LIN {X 0,Y 520.436,Z 843.44,A -85,B 0,C 180,E1 4700.36,E2 4700.36} C_VEL
LIN {X 0,Y 520.239,Z 843.44,A -85,B 0,C 180,E1 4705.948,E2 4705.948} C_VEL
LIN {X 0,Y 520.311,Z 843.44,A -85,B 0,C 180,E1 4711.467,E2 4711.467} C_VEL
LIN {X 0,Y 520.266,Z 843.44,A -85,B 0,C 180,E1 4717.522,E2 4717.522} C_VEL
LIN {X 0,Y 520.062,Z 843.44,A -85,B 0,C 180,E1 4723.497,E2 4723.497} C_VEL
LIN {X 0,Y 520.261,Z 843.44,A -85,B 0,C 180,E1 4730.087,E2 4730.087} C_VEL
LIN {X 0,Y 524.81,Z 853.402,A -85,B 0,C 180,E1 4730.693,E2 4730.693} C_VEL
LIN {X 0,Y 537.138,Z 878.782,A -85,B 0,C 180,E1 4732.342,E2 4732.342} C_VEL
LIN {X 0,Y 535.242,Z 919.42,A -85,B 0,C 180,E1 4733.697,E2 4733.697} C_VEL
LIN {X 0,Y 532.879,Z 957.32,A -85,B 0,C 180,E1 4735.589,E2 4735.589} C_VEL
LIN {X 0,Y 530.11,Z 994.748,A -85,B 0,C 180,E1 4738.147,E2 4738.147} C_VEL
LIN {X 0,Y 527.279,Z 1030.228,A -85,B 0,C 180,E1 4741.356,E2 4741.356} C_VEL
LIN {X 0,Y 524.799,Z 1061.7,A -85,B 0,C 180,E1 4745.046,E2 4745.046} C_VEL
LIN {X 0,Y 522.926,Z 1089.588,A -85,B 0,C 180,E1 4749.298,E2 4749.298} C_VEL
LIN {X 0,Y 521.748,Z 1111.144,A -85,B 0,C 180,E1 4753.621,E2 4753.621} C_VEL
LIN {X 0,Y 521.215,Z 1128.039,A -85,B 0,C 180,E1 4758.307,E2 4758.307} C_VEL
LIN {X 0,Y 520.97,Z 1138.048,A -85,B 0,C 180,E1 4762.51,E2 4762.51} C_VEL
LIN {X 0,Y 520.916,Z 1143.672,A -85,B 0,C 180,E1 4766.678,E2 4766.678} C_VEL
LIN {X 0,Y 521.004,Z 1144.637,A -85,B 0,C 180,E1 4771.66,E2 4771.66} C_VEL
LIN {X 0,Y 520.954,Z 1140.667,A -85,B 0,C 180,E1 4775.819,E2 4775.819} C_VEL
LIN {X 0,Y 521.037,Z 1132.292,A -85,B 0,C 180,E1 4780.049,E2 4780.049} C_VEL
LIN {X 0,Y 521.477,Z 1118.445,A -85,B 0,C 180,E1 4784.459,E2 4784.459} C_VEL
LIN {X 0,Y 522.247,Z 1099.604,A -85,B 0,C 180,E1 4788.751,E2 4788.751} C_VEL
LIN {X 0,Y 523.772,Z 1076.177,A -85,B 0,C 180,E1 4792.795,E2 4792.795} C_VEL
LIN {X 0,Y 525.898,Z 1047.674,A -85,B 0,C 180,E1 4796.619,E2 4796.619} C_VEL
LIN {X 0,Y 528.516,Z 1014.37,A -85,B 0,C 180,E1 4800.095,E2 4800.095} C_VEL
LIN {X 0,Y 531.435,Z 977.699,A -85,B 0,C 180,E1 4803.023,E2 4803.023} C_VEL
LIN {X 0,Y 534.228,Z 938.21,A -85,B 0,C 180,E1 4805.358,E2 4805.358} C_VEL
LIN {X 0,Y 536.423,Z 897.49,A -85,B 0,C 180,E1 4807.024,E2 4807.024} C_VEL
LIN {X 0,Y 536.641,Z 877.029,A -85,B 0,C 180,E1 4807.655,E2 4807.655} C_VEL
LIN {X 0,Y 520.249,Z 844.875,A -85,B 0,C 180,E1 4809.787,E2 4809.787} C_VEL
LIN {X 0,Y 520.083,Z 843.44,A -85,B 0,C 180,E1 4809.907,E2 4809.907} C_VEL
LIN {X 0,Y 520.164,Z 843.44,A -85,B 0,C 180,E1 4815.876,E2 4815.876} C_VEL
LIN {X 0,Y 520.179,Z 843.44,A -85,B 0,C 180,E1 4821.559,E2 4821.559} C_VEL
LIN {X 0,Y 520.166,Z 843.44,A -85,B 0,C 180,E1 4827.277,E2 4827.277} C_VEL
LIN {X 0,Y 520.251,Z 843.44,A -85,B 0,C 180,E1 4832.35,E2 4832.35} C_VEL
LIN {X 0,Y 520.43,Z 843.44,A -85,B 0,C 180,E1 4838.103,E2 4838.103} C_VEL
LIN {X 0,Y 520.561,Z 843.44,A -85,B 0,C 180,E1 4843.15,E2 4843.15} C_VEL
LIN {X 0,Y 520.576,Z 843.44,A -85,B 0,C 180,E1 4848.293,E2 4848.293} C_VEL
LIN {X 0,Y 520.63,Z 843.44,A -85,B 0,C 180,E1 4853.343,E2 4853.343} C_VEL
LIN {X 0,Y 520.641,Z 843.44,A -85,B 0,C 180,E1 4858.339,E2 4858.339} C_VEL
LIN {X 0,Y 520.67,Z 843.44,A -85,B 0,C 180,E1 4863.323,E2 4863.323} C_VEL
LIN {X 0,Y 520.537,Z 843.44,A -85,B 0,C 180,E1 4868.334,E2 4868.334} C_VEL
LIN {X 0,Y 520.491,Z 843.44,A -85,B 0,C 180,E1 4873.411,E2 4873.411} C_VEL
LIN {X 0,Y 520.432,Z 843.44,A -85,B 0,C 180,E1 4878.599,E2 4878.599} C_VEL
LIN {X 0,Y 520.333,Z 843.44,A -85,B 0,C 180,E1 4883.954,E2 4883.954} C_VEL
LIN {X 0,Y 520.209,Z 843.44,A -85,B 0,C 180,E1 4889.546,E2 4889.546} C_VEL
LIN {X 0,Y 520.065,Z 843.44,A -85,B 0,C 180,E1 4894.185,E2 4894.185} C_VEL
LIN {X 0,Y 516.099,Z 843.44,A -85,B 0,C 180,E1 4896.07,E2 4896.07} C_VEL
LIN {X 0,Y 512.255,Z 843.44,A -85,B 0,C 180,E1 4897.985,E2 4897.985} C_VEL
LIN {X 0,Y 512.25,Z 843.44,A -85,B 0,C 180,E1 4902.65,E2 4902.65} C_VEL
LIN {X 0,Y 512.2,Z 843.929,A -85,B 0,C 180,E1 4908.861,E2 4908.861} C_VEL
LIN {X 0,Y 531.6,Z 881.961,A -85,B 0,C 180,E1 4911.305,E2 4911.305} C_VEL
LIN {X 0,Y 530.037,Z 926.984,A -85,B 0,C 180,E1 4912.388,E2 4912.388} C_VEL
LIN {X 0,Y 527.526,Z 969.74,A -85,B 0,C 180,E1 4914.165,E2 4914.165} C_VEL
LIN {X 0,Y 524.424,Z 1009.394,A -85,B 0,C 180,E1 4916.557,E2 4916.557} C_VEL
LIN {X 0,Y 521.221,Z 1047.334,A -85,B 0,C 180,E1 4919.68,E2 4919.68} C_VEL
LIN {X 0,Y 518.367,Z 1080.674,A -85,B 0,C 180,E1 4923.286,E2 4923.286} C_VEL
LIN {X 0,Y 515.864,Z 1110.299,A -85,B 0,C 180,E1 4927.446,E2 4927.446} C_VEL
LIN {X 0,Y 514.329,Z 1134.904,A -85,B 0,C 180,E1 4932.009,E2 4932.009} C_VEL
LIN {X 0,Y 513.485,Z 1152.465,A -85,B 0,C 180,E1 4936.403,E2 4936.403} C_VEL
LIN {X 0,Y 513.102,Z 1164.64,A -85,B 0,C 180,E1 4940.764,E2 4940.764} C_VEL
LIN {X 0,Y 512.92,Z 1171.926,A -85,B 0,C 180,E1 4944.937,E2 4944.937} C_VEL
LIN {X 0,Y 512.92,Z 1174.659,A -85,B 0,C 180,E1 4948.314,E2 4948.314} C_VEL
LIN {X 0,Y 513.175,Z 1174.659,A -85,B 0,C 180,E1 4951.685,E2 4951.685} C_VEL
LIN {X 0,Y 513.034,Z 1169.517,A -85,B 0,C 180,E1 4956.757,E2 4956.757} C_VEL
LIN {X 0,Y 513.348,Z 1159.09,A -85,B 0,C 180,E1 4961.445,E2 4961.445} C_VEL
LIN {X 0,Y 513.978,Z 1142.713,A -85,B 0,C 180,E1 4966.196,E2 4966.196} C_VEL
LIN {X 0,Y 515.2,Z 1121.769,A -85,B 0,C 180,E1 4970.578,E2 4970.578} C_VEL
LIN {X 0,Y 517.007,Z 1095.883,A -85,B 0,C 180,E1 4974.708,E2 4974.708} C_VEL
LIN {X 0,Y 519.533,Z 1066.104,A -85,B 0,C 180,E1 4978.4,E2 4978.4} C_VEL
LIN {X 0,Y 522.495,Z 1031.765,A -85,B 0,C 180,E1 4981.709,E2 4981.709} C_VEL
LIN {X 0,Y 525.589,Z 994.442,A -85,B 0,C 180,E1 4984.44,E2 4984.44} C_VEL
LIN {X 0,Y 528.55,Z 952.967,A -85,B 0,C 180,E1 4986.629,E2 4986.629} C_VEL
LIN {X 0,Y 530.862,Z 909.195,A -85,B 0,C 180,E1 4988.126,E2 4988.126} C_VEL
LIN {X 0,Y 531.26,Z 880.332,A -85,B 0,C 180,E1 4988.755,E2 4988.755} C_VEL
LIN {X 0,Y 512.197,Z 843.964,A -85,B 0,C 180,E1 4991.138,E2 4991.138} C_VEL
LIN {X 0,Y 512.246,Z 843.44,A -85,B 0,C 180,E1 4997.432,E2 4997.432} C_VEL
LIN {X 0,Y 512.233,Z 843.44,A -85,B 0,C 180,E1 5002.694,E2 5002.694} C_VEL
LIN {X 0,Y 512.289,Z 843.44,A -85,B 0,C 180,E1 5008.675,E2 5008.675} C_VEL
LIN {X 0,Y 512.351,Z 843.44,A -85,B 0,C 180,E1 5013.783,E2 5013.783} C_VEL
LIN {X 0,Y 512.551,Z 843.44,A -85,B 0,C 180,E1 5019.312,E2 5019.312} C_VEL
LIN {X 0,Y 512.462,Z 843.44,A -85,B 0,C 180,E1 5024.633,E2 5024.633} C_VEL
LIN {X 0,Y 512.632,Z 843.44,A -85,B 0,C 180,E1 5029.827,E2 5029.827} C_VEL
LIN {X 0,Y 512.845,Z 843.44,A -85,B 0,C 180,E1 5034.936,E2 5034.936} C_VEL
LIN {X 0,Y 512.86,Z 843.44,A -85,B 0,C 180,E1 5040,E2 5040} C_VEL
LIN {X 0,Y 512.812,Z 843.44,A -85,B 0,C 180,E1 5045.064,E2 5045.064} C_VEL
LIN {X 0,Y 512.698,Z 843.44,A -85,B 0,C 180,E1 5050.171,E2 5050.171} C_VEL
LIN {X 0,Y 512.592,Z 843.44,A -85,B 0,C 180,E1 5055.363,E2 5055.363} C_VEL
LIN {X 0,Y 512.532,Z 843.44,A -85,B 0,C 180,E1 5060.689,E2 5060.689} C_VEL
LIN {X 0,Y 512.323,Z 843.44,A -85,B 0,C 180,E1 5066.218,E2 5066.218} C_VEL
LIN {X 0,Y 512.445,Z 843.44,A -85,B 0,C 180,E1 5072.007,E2 5072.007} C_VEL
LIN {X 0,Y 512.324,Z 843.44,A -85,B 0,C 180,E1 5078.208,E2 5078.208} C_VEL
LIN {X 0,Y 512.131,Z 843.44,A -85,B 0,C 180,E1 5085.002,E2 5085.002} C_VEL
LIN {X 0,Y 512.276,Z 843.444,A -85,B 0,C 180,E1 5089.342,E2 5089.342} C_VEL
LIN {X 0,Y 514.638,Z 849.042,A -85,B 0,C 180,E1 5089.67,E2 5089.67} C_VEL
LIN {X 0,Y 530.839,Z 880.706,A -85,B 0,C 180,E1 5091.868,E2 5091.868} C_VEL
LIN {X 0,Y 528.596,Z 923.315,A -85,B 0,C 180,E1 5093.345,E2 5093.345} C_VEL
LIN {X 0,Y 525.764,Z 963.463,A -85,B 0,C 180,E1 5095.463,E2 5095.463} C_VEL
LIN {X 0,Y 522.824,Z 998.946,A -85,B 0,C 180,E1 5098.021,E2 5098.021} C_VEL
LIN {X 0,Y 519.772,Z 1033.362,A -85,B 0,C 180,E1 5101.259,E2 5101.259} C_VEL
LIN {X 0,Y 517.213,Z 1063.294,A -85,B 0,C 180,E1 5104.884,E2 5104.884} C_VEL
LIN {X 0,Y 515.23,Z 1089.586,A -85,B 0,C 180,E1 5108.975,E2 5108.975} C_VEL
LIN {X 0,Y 513.952,Z 1111.142,A -85,B 0,C 180,E1 5113.365,E2 5113.365} C_VEL
LIN {X 0,Y 513.334,Z 1128.036,A -85,B 0,C 180,E1 5118.125,E2 5118.125} C_VEL
LIN {X 0,Y 513.063,Z 1138.047,A -85,B 0,C 180,E1 5122.394,E2 5122.394} C_VEL
LIN {X 0,Y 513.014,Z 1143.671,A -85,B 0,C 180,E1 5126.627,E2 5126.627} C_VEL
LIN {X 0,Y 513.108,Z 1144.638,A -85,B 0,C 180,E1 5131.685,E2 5131.685} C_VEL
LIN {X 0,Y 513.059,Z 1140.668,A -85,B 0,C 180,E1 5135.908,E2 5135.908} C_VEL
LIN {X 0,Y 513.159,Z 1132.409,A -85,B 0,C 180,E1 5140.162,E2 5140.162} C_VEL
LIN {X 0,Y 513.614,Z 1118.479,A -85,B 0,C 180,E1 5144.677,E2 5144.677} C_VEL
LIN {X 0,Y 514.451,Z 1100.693,A -85,B 0,C 180,E1 5148.824,E2 5148.824} C_VEL
LIN {X 0,Y 516.145,Z 1077.203,A -85,B 0,C 180,E1 5152.991,E2 5152.991} C_VEL
LIN {X 0,Y 518.466,Z 1048.615,A -85,B 0,C 180,E1 5156.917,E2 5156.917} C_VEL
LIN {X 0,Y 521.362,Z 1015.638,A -85,B 0,C 180,E1 5160.431,E2 5160.431} C_VEL
LIN {X 0,Y 524.602,Z 978.202,A -85,B 0,C 180,E1 5163.473,E2 5163.473} C_VEL
LIN {X 0,Y 527.627,Z 938.991,A -85,B 0,C 180,E1 5165.826,E2 5165.826} C_VEL
LIN {X 0,Y 530.015,Z 898.735,A -85,B 0,C 180,E1 5167.5,E2 5167.5} C_VEL
LIN {X 0,Y 530.326,Z 880.119,A -85,B 0,C 180,E1 5168.102,E2 5168.102} C_VEL
LIN {X 0,Y 512.171,Z 843.949,A -85,B 0,C 180,E1 5170.568,E2 5170.568} C_VEL
LIN {X 0,Y 512.214,Z 843.44,A -85,B 0,C 180,E1 5175.007,E2 5175.007} C_VEL
LIN {X 0,Y 512.272,Z 843.44,A -85,B 0,C 180,E1 5179.986,E2 5179.986} C_VEL
LIN {X 0,Y 512.175,Z 843.44,A -85,B 0,C 180,E1 5185.96,E2 5185.96} C_VEL
LIN {X 0,Y 512.31,Z 843.44,A -85,B 0,C 180,E1 5192.086,E2 5192.086} C_VEL
LIN {X 0,Y 512.445,Z 843.44,A -85,B 0,C 180,E1 5197.493,E2 5197.493} C_VEL
LIN {X 0,Y 512.652,Z 843.44,A -85,B 0,C 180,E1 5202.882,E2 5202.882} C_VEL
LIN {X 0,Y 512.665,Z 843.44,A -85,B 0,C 180,E1 5208.11,E2 5208.11} C_VEL
LIN {X 0,Y 512.72,Z 843.44,A -85,B 0,C 180,E1 5213.24,E2 5213.24} C_VEL
LIN {X 0,Y 512.741,Z 843.44,A -85,B 0,C 180,E1 5218.314,E2 5218.314} C_VEL
LIN {X 0,Y 512.775,Z 843.44,A -85,B 0,C 180,E1 5223.374,E2 5223.374} C_VEL
LIN {X 0,Y 512.632,Z 843.44,A -85,B 0,C 180,E1 5228.464,E2 5228.464} C_VEL
LIN {X 0,Y 512.577,Z 843.44,A -85,B 0,C 180,E1 5233.709,E2 5233.709} C_VEL
LIN {X 0,Y 512.486,Z 843.44,A -85,B 0,C 180,E1 5239.569,E2 5239.569} C_VEL
LIN {X 0,Y 512.383,Z 843.44,A -85,B 0,C 180,E1 5244.349,E2 5244.349} C_VEL
LIN {X 0,Y 512.246,Z 843.44,A -85,B 0,C 180,E1 5250.052,E2 5250.052} C_VEL
LIN {X 0,Y 512.205,Z 843.44,A -85,B 0,C 180,E1 5256.1,E2 5256.1} C_VEL
LIN {X 0,Y 512.255,Z 843.44,A -85,B 0,C 180,E1 5257.985,E2 5257.985} C_VEL
LIN {X 0,Y 509.802,Z 843.44,A -85,B 0,C 180,E1 5259.415,E2 5259.415} C_VEL
LIN {X 0,Y 504.24,Z 843.44,A -85,B 0,C 180,E1 5261.805,E2 5261.805} C_VEL
LIN {X 0,Y 504.315,Z 844.166,A -85,B 0,C 180,E1 5268.086,E2 5268.086} C_VEL
LIN {X 0,Y 525.368,Z 884.453,A -85,B 0,C 180,E1 5270.809,E2 5270.809} C_VEL
LIN {X 0,Y 523.699,Z 927.636,A -85,B 0,C 180,E1 5271.878,E2 5271.878} C_VEL
LIN {X 0,Y 521.018,Z 969.675,A -85,B 0,C 180,E1 5273.643,E2 5273.643} C_VEL
LIN {X 0,Y 517.667,Z 1009.395,A -85,B 0,C 180,E1 5276.062,E2 5276.062} C_VEL
LIN {X 0,Y 514.143,Z 1047.323,A -85,B 0,C 180,E1 5279.217,E2 5279.217} C_VEL
LIN {X 0,Y 510.953,Z 1081.461,A -85,B 0,C 180,E1 5282.973,E2 5282.973} C_VEL
LIN {X 0,Y 508.335,Z 1110.222,A -85,B 0,C 180,E1 5287.079,E2 5287.079} C_VEL
LIN {X 0,Y 506.689,Z 1134.088,A -85,B 0,C 180,E1 5291.542,E2 5291.542} C_VEL
LIN {X 0,Y 505.667,Z 1152.464,A -85,B 0,C 180,E1 5296.188,E2 5296.188} C_VEL
LIN {X 0,Y 505.21,Z 1165.116,A -85,B 0,C 180,E1 5300.834,E2 5300.834} C_VEL
LIN {X 0,Y 505.022,Z 1171.926,A -85,B 0,C 180,E1 5304.857,E2 5304.857} C_VEL
LIN {X 0,Y 505.018,Z 1174.659,A -85,B 0,C 180,E1 5308.288,E2 5308.288} C_VEL
LIN {X 0,Y 505.27,Z 1174.659,A -85,B 0,C 180,E1 5311.712,E2 5311.712} C_VEL
LIN {X 0,Y 505.137,Z 1169.517,A -85,B 0,C 180,E1 5316.863,E2 5316.863} C_VEL
LIN {X 0,Y 505.471,Z 1159.091,A -85,B 0,C 180,E1 5321.626,E2 5321.626} C_VEL
LIN {X 0,Y 506.178,Z 1142.714,A -85,B 0,C 180,E1 5326.452,E2 5326.452} C_VEL
LIN {X 0,Y 507.529,Z 1121.768,A -85,B 0,C 180,E1 5330.903,E2 5330.903} C_VEL
LIN {X 0,Y 509.494,Z 1096.45,A -85,B 0,C 180,E1 5335.014,E2 5335.014} C_VEL
LIN {X 0,Y 512.269,Z 1066.678,A -85,B 0,C 180,E1 5338.774,E2 5338.774} C_VEL
LIN {X 0,Y 515.521,Z 1032.556,A -85,B 0,C 180,E1 5342.118,E2 5342.118} C_VEL
LIN {X 0,Y 518.902,Z 994.749,A -85,B 0,C 180,E1 5344.927,E2 5344.927} C_VEL
LIN {X 0,Y 522.128,Z 953.443,A -85,B 0,C 180,E1 5347.133,E2 5347.133} C_VEL
LIN {X 0,Y 524.58,Z 911.065,A -85,B 0,C 180,E1 5348.614,E2 5348.614} C_VEL
LIN {X 0,Y 525.023,Z 883.051,A -85,B 0,C 180,E1 5349.25,E2 5349.25} C_VEL
LIN {X 0,Y 504.318,Z 844.136,A -85,B 0,C 180,E1 5351.914,E2 5351.914} C_VEL
LIN {X 0,Y 504.266,Z 843.44,A -85,B 0,C 180,E1 5358.428,E2 5358.428} C_VEL
LIN {X 0,Y 504.343,Z 843.44,A -85,B 0,C 180,E1 5363.887,E2 5363.887} C_VEL
LIN {X 0,Y 504.327,Z 843.44,A -85,B 0,C 180,E1 5370.195,E2 5370.195} C_VEL
LIN {X 0,Y 504.428,Z 843.44,A -85,B 0,C 180,E1 5375.241,E2 5375.241} C_VEL
LIN {X 0,Y 504.669,Z 843.44,A -85,B 0,C 180,E1 5380.798,E2 5380.798} C_VEL
LIN {X 0,Y 504.482,Z 843.44,A -85,B 0,C 180,E1 5386.155,E2 5386.155} C_VEL
LIN {X 0,Y 504.712,Z 843.44,A -85,B 0,C 180,E1 5391.403,E2 5391.403} C_VEL
LIN {X 0,Y 504.875,Z 843.44,A -85,B 0,C 180,E1 5396.573,E2 5396.573} C_VEL
LIN {X 0,Y 504.845,Z 843.44,A -85,B 0,C 180,E1 5401.713,E2 5401.713} C_VEL
LIN {X 0,Y 504.804,Z 843.44,A -85,B 0,C 180,E1 5406.867,E2 5406.867} C_VEL
LIN {X 0,Y 504.723,Z 843.44,A -85,B 0,C 180,E1 5412.08,E2 5412.08} C_VEL
LIN {X 0,Y 504.677,Z 843.44,A -85,B 0,C 180,E1 5417.397,E2 5417.397} C_VEL
LIN {X 0,Y 504.507,Z 843.44,A -85,B 0,C 180,E1 5422.881,E2 5422.881} C_VEL
LIN {X 0,Y 504.393,Z 843.44,A -85,B 0,C 180,E1 5428.598,E2 5428.598} C_VEL
LIN {X 0,Y 504.487,Z 843.44,A -85,B 0,C 180,E1 5434.632,E2 5434.632} C_VEL
LIN {X 0,Y 504.225,Z 843.44,A -85,B 0,C 180,E1 5441.176,E2 5441.176} C_VEL
LIN {X 0,Y 504.16,Z 843.44,A -85,B 0,C 180,E1 5446.495,E2 5446.495} C_VEL
LIN {X 0,Y 504.287,Z 843.585,A -85,B 0,C 180,E1 5448.555,E2 5448.555} C_VEL
LIN {X 0,Y 508.488,Z 852.603,A -85,B 0,C 180,E1 5449.143,E2 5449.143} C_VEL
LIN {X 0,Y 524.313,Z 883.255,A -85,B 0,C 180,E1 5451.391,E2 5451.391} C_VEL
LIN {X 0,Y 522.069,Z 925.289,A -85,B 0,C 180,E1 5452.909,E2 5452.909} C_VEL
LIN {X 0,Y 518.814,Z 967.192,A -85,B 0,C 180,E1 5455.193,E2 5455.193} C_VEL
LIN {X 0,Y 515.224,Z 1006.042,A -85,B 0,C 180,E1 5458.139,E2 5458.139} C_VEL
LIN {X 0,Y 511.93,Z 1040.776,A -85,B 0,C 180,E1 5461.641,E2 5461.641} C_VEL
LIN {X 0,Y 509.114,Z 1071.581,A -85,B 0,C 180,E1 5465.688,E2 5465.688} C_VEL
LIN {X 0,Y 507.049,Z 1097.701,A -85,B 0,C 180,E1 5470.181,E2 5470.181} C_VEL
LIN {X 0,Y 505.926,Z 1117.481,A -85,B 0,C 180,E1 5474.719,E2 5474.719} C_VEL
LIN {X 0,Y 505.31,Z 1132.641,A -85,B 0,C 180,E1 5479.678,E2 5479.678} C_VEL
LIN {X 0,Y 505.091,Z 1140.795,A -85,B 0,C 180,E1 5483.998,E2 5483.998} C_VEL
LIN {X 0,Y 505.025,Z 1144.675,A -85,B 0,C 180,E1 5488.288,E2 5488.288} C_VEL
LIN {X 0,Y 505.202,Z 1144.638,A -85,B 0,C 180,E1 5491.711,E2 5491.711} C_VEL
LIN {X 0,Y 505.165,Z 1140.668,A -85,B 0,C 180,E1 5496.001,E2 5496.001} C_VEL
LIN {X 0,Y 505.276,Z 1132.411,A -85,B 0,C 180,E1 5500.322,E2 5500.322} C_VEL
LIN {X 0,Y 505.793,Z 1118.22,A -85,B 0,C 180,E1 5504.984,E2 5504.984} C_VEL
LIN {X 0,Y 506.723,Z 1100.695,A -85,B 0,C 180,E1 5509.122,E2 5509.122} C_VEL
LIN {X 0,Y 508.535,Z 1077.437,A -85,B 0,C 180,E1 5513.319,E2 5513.319} C_VEL
LIN {X 0,Y 511.181,Z 1047.883,A -85,B 0,C 180,E1 5517.425,E2 5517.425} C_VEL
LIN {X 0,Y 514.461,Z 1014.39,A -85,B 0,C 180,E1 5521.007,E2 5521.007} C_VEL
LIN {X 0,Y 517.927,Z 977.123,A -85,B 0,C 180,E1 5524.045,E2 5524.045} C_VEL
LIN {X 0,Y 521.224,Z 937.756,A -85,B 0,C 180,E1 5526.405,E2 5526.405} C_VEL
LIN {X 0,Y 523.809,Z 897.766,A -85,B 0,C 180,E1 5528.062,E2 5528.062} C_VEL
LIN {X 0,Y 523.988,Z 883.073,A -85,B 0,C 180,E1 5528.553,E2 5528.553} C_VEL
LIN {X 0,Y 504.309,Z 844.705,A -85,B 0,C 180,E1 5531.332,E2 5531.332} C_VEL
LIN {X 0,Y 504.227,Z 843.44,A -85,B 0,C 180,E1 5531.404,E2 5531.404} C_VEL
LIN {X 0,Y 504.232,Z 843.44,A -85,B 0,C 180,E1 5536.505,E2 5536.505} C_VEL
LIN {X 0,Y 504.326,Z 843.44,A -85,B 0,C 180,E1 5541.074,E2 5541.074} C_VEL
LIN {X 0,Y 504.262,Z 843.44,A -85,B 0,C 180,E1 5547.41,E2 5547.41} C_VEL
LIN {X 0,Y 504.434,Z 843.44,A -85,B 0,C 180,E1 5553.825,E2 5553.825} C_VEL
LIN {X 0,Y 504.603,Z 843.44,A -85,B 0,C 180,E1 5558.971,E2 5558.971} C_VEL
LIN {X 0,Y 504.748,Z 843.44,A -85,B 0,C 180,E1 5564.392,E2 5564.392} C_VEL
LIN {X 0,Y 504.775,Z 843.44,A -85,B 0,C 180,E1 5570.584,E2 5570.584} C_VEL
LIN {X 0,Y 505.018,Z 843.44,A -85,B 0,C 180,E1 5576.574,E2 5576.574} C_VEL
LIN {X 0,Y 505.117,Z 843.44,A -85,B 0,C 180,E1 5581.712,E2 5581.712} C_VEL
LIN {X 0,Y 504.887,Z 843.44,A -85,B 0,C 180,E1 5586.866,E2 5586.866} C_VEL
LIN {X 0,Y 504.71,Z 843.44,A -85,B 0,C 180,E1 5592.08,E2 5592.08} C_VEL
LIN {X 0,Y 504.634,Z 843.44,A -85,B 0,C 180,E1 5597.399,E2 5597.399} C_VEL
LIN {X 0,Y 504.495,Z 843.44,A -85,B 0,C 180,E1 5602.882,E2 5602.882} C_VEL
LIN {X 0,Y 504.363,Z 843.44,A -85,B 0,C 180,E1 5608.6,E2 5608.6} C_VEL
LIN {X 0,Y 504.27,Z 843.44,A -85,B 0,C 180,E1 5614.649,E2 5614.649} C_VEL
LIN {X 0,Y 504.286,Z 843.44,A -85,B 0,C 180,E1 5621.17,E2 5621.17} C_VEL
LIN {X 0,Y 504.24,Z 843.44,A -85,B 0,C 180,E1 5621.805,E2 5621.805} C_VEL
LIN {X 0,Y 500.248,Z 843.44,A -85,B 0,C 180,E1 5623.754,E2 5623.754} C_VEL
LIN {X 0,Y 496.309,Z 843.44,A -85,B 0,C 180,E1 5625.732,E2 5625.732} C_VEL
LIN {X 0,Y 496.36,Z 843.44,A -85,B 0,C 180,E1 5627.23,E2 5627.23} C_VEL
LIN {X 0,Y 500.68,Z 852.873,A -85,B 0,C 180,E1 5627.879,E2 5627.879} C_VEL
LIN {X 0,Y 519.189,Z 886.645,A -85,B 0,C 180,E1 5630.297,E2 5630.297} C_VEL
LIN {X 0,Y 517.346,Z 929.486,A -85,B 0,C 180,E1 5631.4,E2 5631.4} C_VEL
LIN {X 0,Y 514.459,Z 970.757,A -85,B 0,C 180,E1 5633.17,E2 5633.17} C_VEL
LIN {X 0,Y 510.866,Z 1010.222,A -85,B 0,C 180,E1 5635.615,E2 5635.615} C_VEL
LIN {X 0,Y 507.025,Z 1048.058,A -85,B 0,C 180,E1 5638.816,E2 5638.816} C_VEL
LIN {X 0,Y 503.561,Z 1082.165,A -85,B 0,C 180,E1 5642.64,E2 5642.64} C_VEL
LIN {X 0,Y 500.669,Z 1111.503,A -85,B 0,C 180,E1 5646.932,E2 5646.932} C_VEL
LIN {X 0,Y 498.866,Z 1135.122,A -85,B 0,C 180,E1 5651.482,E2 5651.482} C_VEL
LIN {X 0,Y 497.845,Z 1152.463,A -85,B 0,C 180,E1 5655.967,E2 5655.967} C_VEL
LIN {X 0,Y 497.339,Z 1165.116,A -85,B 0,C 180,E1 5660.687,E2 5660.687} C_VEL
LIN {X 0,Y 497.129,Z 1171.926,A -85,B 0,C 180,E1 5664.775,E2 5664.775} C_VEL
LIN {X 0,Y 497.116,Z 1174.659,A -85,B 0,C 180,E1 5668.261,E2 5668.261} C_VEL
LIN {X 0,Y 497.38,Z 1174.659,A -85,B 0,C 180,E1 5671.739,E2 5671.739} C_VEL
LIN {X 0,Y 497.246,Z 1169.517,A -85,B 0,C 180,E1 5676.973,E2 5676.973} C_VEL
LIN {X 0,Y 497.593,Z 1159.092,A -85,B 0,C 180,E1 5681.812,E2 5681.812} C_VEL
LIN {X 0,Y 498.373,Z 1142.716,A -85,B 0,C 180,E1 5686.717,E2 5686.717} C_VEL
LIN {X 0,Y 499.845,Z 1121.766,A -85,B 0,C 180,E1 5691.24,E2 5691.24} C_VEL
LIN {X 0,Y 502.127,Z 1095.85,A -85,B 0,C 180,E1 5695.497,E2 5695.497} C_VEL
LIN {X 0,Y 505.19,Z 1065.52,A -85,B 0,C 180,E1 5699.352,E2 5699.352} C_VEL
LIN {X 0,Y 508.683,Z 1032.016,A -85,B 0,C 180,E1 5702.652,E2 5702.652} C_VEL
LIN {X 0,Y 512.396,Z 993.619,A -85,B 0,C 180,E1 5705.515,E2 5705.515} C_VEL
LIN {X 0,Y 515.79,Z 953.429,A -85,B 0,C 180,E1 5707.669,E2 5707.669} C_VEL
LIN {X 0,Y 518.472,Z 909.512,A -85,B 0,C 180,E1 5709.2,E2 5709.2} C_VEL
LIN {X 0,Y 518.709,Z 885.753,A -85,B 0,C 180,E1 5709.765,E2 5709.765} C_VEL
LIN {X 0,Y 496.486,Z 844.831,A -85,B 0,C 180,E1 5712.71,E2 5712.71} C_VEL
LIN {X 0,Y 496.36,Z 843.44,A -85,B 0,C 180,E1 5712.845,E2 5712.845} C_VEL
LIN {X 0,Y 496.321,Z 843.44,A -85,B 0,C 180,E1 5718.021,E2 5718.021} C_VEL
LIN {X 0,Y 496.379,Z 843.44,A -85,B 0,C 180,E1 5724.719,E2 5724.719} C_VEL
LIN {X 0,Y 496.428,Z 843.44,A -85,B 0,C 180,E1 5730.9,E2 5730.9} C_VEL
LIN {X 0,Y 496.541,Z 843.44,A -85,B 0,C 180,E1 5736.73,E2 5736.73} C_VEL
LIN {X 0,Y 496.767,Z 843.44,A -85,B 0,C 180,E1 5742.317,E2 5742.317} C_VEL
LIN {X 0,Y 496.779,Z 843.44,A -85,B 0,C 180,E1 5749.499,E2 5749.499} C_VEL
LIN {X 0,Y 497.034,Z 843.44,A -85,B 0,C 180,E1 5754.774,E2 5754.774} C_VEL
LIN {X 0,Y 497.066,Z 843.44,A -85,B 0,C 180,E1 5760,E2 5760} C_VEL
LIN {X 0,Y 496.998,Z 843.44,A -85,B 0,C 180,E1 5765.226,E2 5765.226} C_VEL
LIN {X 0,Y 496.862,Z 843.44,A -85,B 0,C 180,E1 5770.499,E2 5770.499} C_VEL
LIN {X 0,Y 496.752,Z 843.44,A -85,B 0,C 180,E1 5775.866,E2 5775.866} C_VEL
LIN {X 0,Y 496.65,Z 843.44,A -85,B 0,C 180,E1 5781.382,E2 5781.382} C_VEL
LIN {X 0,Y 496.453,Z 843.44,A -85,B 0,C 180,E1 5787.124,E2 5787.124} C_VEL
LIN {X 0,Y 496.556,Z 843.44,A -85,B 0,C 180,E1 5793.161,E2 5793.161} C_VEL
LIN {X 0,Y 496.352,Z 843.44,A -85,B 0,C 180,E1 5799.674,E2 5799.674} C_VEL
LIN {X 0,Y 496.237,Z 843.44,A -85,B 0,C 180,E1 5805.62,E2 5805.62} C_VEL
LIN {X 0,Y 496.296,Z 843.44,A -85,B 0,C 180,E1 5807.709,E2 5807.709} C_VEL
LIN {X 0,Y 498.826,Z 849.175,A -85,B 0,C 180,E1 5808.101,E2 5808.101} C_VEL
LIN {X 0,Y 517.933,Z 886.118,A -85,B 0,C 180,E1 5810.924,E2 5810.924} C_VEL
LIN {X 0,Y 515.588,Z 926.528,A -85,B 0,C 180,E1 5812.431,E2 5812.431} C_VEL
LIN {X 0,Y 512.245,Z 966.564,A -85,B 0,C 180,E1 5814.634,E2 5814.634} C_VEL
LIN {X 0,Y 508.414,Z 1005.256,A -85,B 0,C 180,E1 5817.583,E2 5817.583} C_VEL
LIN {X 0,Y 504.691,Z 1040.94,A -85,B 0,C 180,E1 5821.219,E2 5821.219} C_VEL
LIN {X 0,Y 501.599,Z 1071.754,A -85,B 0,C 180,E1 5825.328,E2 5825.328} C_VEL
LIN {X 0,Y 499.447,Z 1096.508,A -85,B 0,C 180,E1 5829.616,E2 5829.616} C_VEL
LIN {X 0,Y 498.163,Z 1116.36,A -85,B 0,C 180,E1 5834.179,E2 5834.179} C_VEL
LIN {X 0,Y 497.497,Z 1131.501,A -85,B 0,C 180,E1 5839.072,E2 5839.072} C_VEL
LIN {X 0,Y 497.231,Z 1139.586,A -85,B 0,C 180,E1 5843.027,E2 5843.027} C_VEL
LIN {X 0,Y 497.207,Z 1143.67,A -85,B 0,C 180,E1 5846.52,E2 5846.52} C_VEL
LIN {X 0,Y 497.296,Z 1144.639,A -85,B 0,C 180,E1 5851.739,E2 5851.739} C_VEL
LIN {X 0,Y 497.257,Z 1140.669,A -85,B 0,C 180,E1 5856.097,E2 5856.097} C_VEL
LIN {X 0,Y 497.382,Z 1132.412,A -85,B 0,C 180,E1 5860.488,E2 5860.488} C_VEL
LIN {X 0,Y 498.002,Z 1117.708,A -85,B 0,C 180,E1 5865.374,E2 5865.374} C_VEL
LIN {X 0,Y 499.265,Z 1098.01,A -85,B 0,C 180,E1 5869.987,E2 5869.987} C_VEL
LIN {X 0,Y 501.513,Z 1072.667,A -85,B 0,C 180,E1 5874.439,E2 5874.439} C_VEL
LIN {X 0,Y 504.374,Z 1043.677,A -85,B 0,C 180,E1 5878.362,E2 5878.362} C_VEL
LIN {X 0,Y 507.811,Z 1010.756,A -85,B 0,C 180,E1 5881.821,E2 5881.821} C_VEL
LIN {X 0,Y 511.322,Z 976.201,A -85,B 0,C 180,E1 5884.617,E2 5884.617} C_VEL
LIN {X 0,Y 514.775,Z 937.841,A -85,B 0,C 180,E1 5886.932,E2 5886.932} C_VEL
LIN {X 0,Y 517.534,Z 898.37,A -85,B 0,C 180,E1 5888.584,E2 5888.584} C_VEL
LIN {X 0,Y 517.651,Z 886.086,A -85,B 0,C 180,E1 5889.012,E2 5889.012} C_VEL
LIN {X 0,Y 498.819,Z 849.224,A -85,B 0,C 180,E1 5891.809,E2 5891.809} C_VEL
LIN {X 0,Y 496.227,Z 843.44,A -85,B 0,C 180,E1 5892.287,E2 5892.287} C_VEL
LIN {X 0,Y 496.302,Z 843.44,A -85,B 0,C 180,E1 5898.019,E2 5898.019} C_VEL
LIN {X 0,Y 496.367,Z 843.44,A -85,B 0,C 180,E1 5904.718,E2 5904.718} C_VEL
LIN {X 0,Y 496.417,Z 843.44,A -85,B 0,C 180,E1 5910.899,E2 5910.899} C_VEL
LIN {X 0,Y 496.539,Z 843.44,A -85,B 0,C 180,E1 5916.73,E2 5916.73} C_VEL
LIN {X 0,Y 496.776,Z 843.44,A -85,B 0,C 180,E1 5922.317,E2 5922.317} C_VEL
LIN {X 0,Y 496.844,Z 843.44,A -85,B 0,C 180,E1 5927.726,E2 5927.726} C_VEL
LIN {X 0,Y 496.924,Z 843.44,A -85,B 0,C 180,E1 5933.024,E2 5933.024} C_VEL
LIN {X 0,Y 496.964,Z 843.44,A -85,B 0,C 180,E1 5938.26,E2 5938.26} C_VEL
LIN {X 0,Y 496.986,Z 843.44,A -85,B 0,C 180,E1 5943.482,E2 5943.482} C_VEL
LIN {X 0,Y 496.824,Z 843.44,A -85,B 0,C 180,E1 5948.735,E2 5948.735} C_VEL
LIN {X 0,Y 496.767,Z 843.44,A -85,B 0,C 180,E1 5954.064,E2 5954.064} C_VEL
LIN {X 0,Y 496.64,Z 843.44,A -85,B 0,C 180,E1 5959.624,E2 5959.624} C_VEL
LIN {X 0,Y 496.528,Z 843.44,A -85,B 0,C 180,E1 5965.18,E2 5965.18} C_VEL
LIN {X 0,Y 496.321,Z 843.44,A -85,B 0,C 180,E1 5971.646,E2 5971.646} C_VEL
LIN {X 0,Y 496.32,Z 843.44,A -85,B 0,C 180,E1 5977.768,E2 5977.768} C_VEL
LIN {X 0,Y 496.339,Z 843.44,A -85,B 0,C 180,E1 5984.366,E2 5984.366} C_VEL
LIN {X 0,Y 496.309,Z 843.44,A -85,B 0,C 180,E1 5985.732,E2 5985.732} C_VEL
LIN {X 0,Y 496.515,Z 846.56,A -85,B 0,C 180,E1 5986.618,E2 5986.618} C_VEL
LIN {X 0,Y 498.004,Z 857.238,A -85,B 0,C 180,E1 5987.561,E2 5987.561} C_VEL
LIN {X 0,Y 502.24,Z 869.127,A -85,B 0,C 180,E1 5988.343,E2 5988.343} C_VEL
LIN {X 0,Y 512.968,Z 889.52,A -85,B 0,C 180,E1 5989.786,E2 5989.786} C_VEL
LIN {X 0,Y 511.021,Z 931.258,A -85,B 0,C 180,E1 5990.91,E2 5990.91} C_VEL
LIN {X 0,Y 507.989,Z 971.227,A -85,B 0,C 180,E1 5992.651,E2 5992.651} C_VEL
LIN {X 0,Y 504.009,Z 1011.681,A -85,B 0,C 180,E1 5995.204,E2 5995.204} C_VEL
LIN {X 0,Y 500.106,Z 1047.572,A -85,B 0,C 180,E1 5998.282,E2 5998.282} C_VEL
LIN {X 0,Y 496.283,Z 1081.676,A -85,B 0,C 180,E1 6002.136,E2 6002.136} C_VEL
LIN {X 0,Y 493.282,Z 1110.168,A -85,B 0,C 180,E1 6006.327,E2 6006.327} C_VEL
LIN {X 0,Y 491.224,Z 1134.139,A -85,B 0,C 180,E1 6010.95,E2 6010.95} C_VEL
LIN {X 0,Y 490.037,Z 1152.462,A -85,B 0,C 180,E1 6015.738,E2 6015.738} C_VEL
LIN {X 0,Y 489.447,Z 1165.24,A -85,B 0,C 180,E1 6020.594,E2 6020.594} C_VEL
LIN {X 0,Y 489.233,Z 1171.926,A -85,B 0,C 180,E1 6024.691,E2 6024.691} C_VEL
LIN {X 0,Y 489.214,Z 1174.659,A -85,B 0,C 180,E1 6028.233,E2 6028.233} C_VEL
LIN {X 0,Y 489.474,Z 1174.659,A -85,B 0,C 180,E1 6031.767,E2 6031.767} C_VEL
LIN {X 0,Y 489.349,Z 1169.517,A -85,B 0,C 180,E1 6037.086,E2 6037.086} C_VEL
LIN {X 0,Y 489.72,Z 1159.092,A -85,B 0,C 180,E1 6042.005,E2 6042.005} C_VEL
LIN {X 0,Y 490.561,Z 1143.355,A -85,B 0,C 180,E1 6046.824,E2 6046.824} C_VEL
LIN {X 0,Y 492.107,Z 1122.841,A -85,B 0,C 180,E1 6051.379,E2 6051.379} C_VEL
LIN {X 0,Y 494.561,Z 1097.332,A -85,B 0,C 180,E1 6055.69,E2 6055.69} C_VEL
LIN {X 0,Y 497.806,Z 1067.903,A -85,B 0,C 180,E1 6059.546,E2 6059.546} C_VEL
LIN {X 0,Y 501.774,Z 1032.527,A -85,B 0,C 180,E1 6063.112,E2 6063.112} C_VEL
LIN {X 0,Y 505.741,Z 994.713,A -85,B 0,C 180,E1 6065.978,E2 6065.978} C_VEL
LIN {X 0,Y 509.493,Z 953.43,A -85,B 0,C 180,E1 6068.218,E2 6068.218} C_VEL
LIN {X 0,Y 512.333,Z 909.284,A -85,B 0,C 180,E1 6069.762,E2 6069.762} C_VEL
LIN {X 0,Y 512.56,Z 888.801,A -85,B 0,C 180,E1 6070.268,E2 6070.268} C_VEL
LIN {X 0,Y 490.006,Z 848.156,A -85,B 0,C 180,E1 6073.342,E2 6073.342} C_VEL
LIN {X 0,Y 488.401,Z 843.44,A -85,B 0,C 180,E1 6073.66,E2 6073.66} C_VEL
LIN {X 0,Y 488.421,Z 843.44,A -85,B 0,C 180,E1 6079.55,E2 6079.55} C_VEL
LIN {X 0,Y 488.439,Z 843.44,A -85,B 0,C 180,E1 6086.215,E2 6086.215} C_VEL
LIN {X 0,Y 488.519,Z 843.44,A -85,B 0,C 180,E1 6092.398,E2 6092.398} C_VEL
LIN {X 0,Y 488.697,Z 843.44,A -85,B 0,C 180,E1 6098.252,E2 6098.252} C_VEL
LIN {X 0,Y 488.758,Z 843.44,A -85,B 0,C 180,E1 6103.867,E2 6103.867} C_VEL
LIN {X 0,Y 488.856,Z 843.44,A -85,B 0,C 180,E1 6109.327,E2 6109.327} C_VEL
LIN {X 0,Y 489.121,Z 843.44,A -85,B 0,C 180,E1 6114.689,E2 6114.689} C_VEL
LIN {X 0,Y 489.165,Z 843.44,A -85,B 0,C 180,E1 6120,E2 6120} C_VEL
LIN {X 0,Y 489.083,Z 843.44,A -85,B 0,C 180,E1 6125.311,E2 6125.311} C_VEL
LIN {X 0,Y 488.936,Z 843.44,A -85,B 0,C 180,E1 6130.671,E2 6130.671} C_VEL
LIN {X 0,Y 488.784,Z 843.44,A -85,B 0,C 180,E1 6136.851,E2 6136.851} C_VEL
LIN {X 0,Y 488.673,Z 843.44,A -85,B 0,C 180,E1 6142.12,E2 6142.12} C_VEL
LIN {X 0,Y 488.536,Z 843.44,A -85,B 0,C 180,E1 6147.601,E2 6147.601} C_VEL
LIN {X 0,Y 488.614,Z 843.44,A -85,B 0,C 180,E1 6153.771,E2 6153.771} C_VEL
LIN {X 0,Y 488.435,Z 843.44,A -85,B 0,C 180,E1 6159.432,E2 6159.432} C_VEL
LIN {X 0,Y 488.331,Z 843.44,A -85,B 0,C 180,E1 6165.292,E2 6165.292} C_VEL
LIN {X 0,Y 488.371,Z 843.44,A -85,B 0,C 180,E1 6166.84,E2 6166.84} C_VEL
LIN {X 0,Y 490.891,Z 849.214,A -85,B 0,C 180,E1 6167.258,E2 6167.258} C_VEL
LIN {X 0,Y 510.151,Z 885.647,A -85,B 0,C 180,E1 6170.185,E2 6170.185} C_VEL
LIN {X 0,Y 511.746,Z 890.75,A -85,B 0,C 180,E1 6170.515,E2 6170.515} C_VEL
LIN {X 0,Y 508.956,Z 929.535,A -85,B 0,C 180,E1 6172.023,E2 6172.023} C_VEL
LIN {X 0,Y 505.396,Z 969.044,A -85,B 0,C 180,E1 6174.275,E2 6174.275} C_VEL
LIN {X 0,Y 501.385,Z 1006.478,A -85,B 0,C 180,E1 6177.197,E2 6177.197} C_VEL
LIN {X 0,Y 497.437,Z 1041.136,A -85,B 0,C 180,E1 6180.785,E2 6180.785} C_VEL
LIN {X 0,Y 494.124,Z 1071.751,A -85,B 0,C 180,E1 6184.929,E2 6184.929} C_VEL
LIN {X 0,Y 491.681,Z 1097.666,A -85,B 0,C 180,E1 6189.527,E2 6189.527} C_VEL
LIN {X 0,Y 490.274,Z 1118.012,A -85,B 0,C 180,E1 6194.376,E2 6194.376} C_VEL
LIN {X 0,Y 489.577,Z 1132.637,A -85,B 0,C 180,E1 6199.342,E2 6199.342} C_VEL
LIN {X 0,Y 489.3,Z 1140.792,A -85,B 0,C 180,E1 6203.803,E2 6203.803} C_VEL
LIN {X 0,Y 489.221,Z 1144.675,A -85,B 0,C 180,E1 6208.232,E2 6208.232} C_VEL
LIN {X 0,Y 489.39,Z 1144.639,A -85,B 0,C 180,E1 6211.767,E2 6211.767} C_VEL
LIN {X 0,Y 489.347,Z 1140.67,A -85,B 0,C 180,E1 6216.196,E2 6216.196} C_VEL
LIN {X 0,Y 489.516,Z 1132.414,A -85,B 0,C 180,E1 6220.659,E2 6220.659} C_VEL
LIN {X 0,Y 490.102,Z 1119.254,A -85,B 0,C 180,E1 6225.172,E2 6225.172} C_VEL
LIN {X 0,Y 491.229,Z 1101.781,A -85,B 0,C 180,E1 6229.516,E2 6229.516} C_VEL
LIN {X 0,Y 493.401,Z 1078.489,A -85,B 0,C 180,E1 6233.906,E2 6233.906} C_VEL
LIN {X 0,Y 496.62,Z 1048.52,A -85,B 0,C 180,E1 6238.219,E2 6238.219} C_VEL
LIN {X 0,Y 500.374,Z 1015.549,A -85,B 0,C 180,E1 6241.865,E2 6241.865} C_VEL
LIN {X 0,Y 504.476,Z 978.114,A -85,B 0,C 180,E1 6245.008,E2 6245.008} C_VEL
LIN {X 0,Y 508.401,Z 937.767,A -85,B 0,C 180,E1 6247.479,E2 6247.479} C_VEL
LIN {X 0,Y 511.347,Z 898.929,A -85,B 0,C 180,E1 6249.123,E2 6249.123} C_VEL
LIN {X 0,Y 511.28,Z 888.929,A -85,B 0,C 180,E1 6249.503,E2 6249.503} C_VEL
LIN {X 0,Y 493.856,Z 854.553,A -85,B 0,C 180,E1 6252.221,E2 6252.221} C_VEL
LIN {X 0,Y 488.387,Z 844.171,A -85,B 0,C 180,E1 6253.026,E2 6253.026} C_VEL
LIN {X 0,Y 488.397,Z 843.44,A -85,B 0,C 180,E1 6257.862,E2 6257.862} C_VEL
LIN {X 0,Y 488.378,Z 843.44,A -85,B 0,C 180,E1 6264.052,E2 6264.052} C_VEL
LIN {X 0,Y 488.442,Z 843.44,A -85,B 0,C 180,E1 6270.377,E2 6270.377} C_VEL
LIN {X 0,Y 488.636,Z 843.44,A -85,B 0,C 180,E1 6276.331,E2 6276.331} C_VEL
LIN {X 0,Y 488.845,Z 843.44,A -85,B 0,C 180,E1 6282.021,E2 6282.021} C_VEL
LIN {X 0,Y 488.97,Z 843.44,A -85,B 0,C 180,E1 6287.525,E2 6287.525} C_VEL
LIN {X 0,Y 489.01,Z 843.44,A -85,B 0,C 180,E1 6292.91,E2 6292.91} C_VEL
LIN {X 0,Y 489.064,Z 843.44,A -85,B 0,C 180,E1 6298.232,E2 6298.232} C_VEL
LIN {X 0,Y 489.08,Z 843.44,A -85,B 0,C 180,E1 6303.538,E2 6303.538} C_VEL
LIN {X 0,Y 488.914,Z 843.44,A -85,B 0,C 180,E1 6309.008,E2 6309.008} C_VEL
LIN {X 0,Y 488.829,Z 843.44,A -85,B 0,C 180,E1 6314.297,E2 6314.297} C_VEL
LIN {X 0,Y 488.731,Z 843.44,A -85,B 0,C 180,E1 6319.854,E2 6319.854} C_VEL
LIN {X 0,Y 488.565,Z 843.44,A -85,B 0,C 180,E1 6325.62,E2 6325.62} C_VEL
LIN {X 0,Y 488.418,Z 843.44,A -85,B 0,C 180,E1 6331.683,E2 6331.683} C_VEL
LIN {X 0,Y 488.403,Z 843.44,A -85,B 0,C 180,E1 6338.164,E2 6338.164} C_VEL
LIN {X 0,Y 488.417,Z 843.44,A -85,B 0,C 180,E1 6344.716,E2 6344.716} C_VEL
LIN {X 0,Y 488.426,Z 843.44,A -85,B 0,C 180,E1 6346.378,E2 6346.378} C_VEL
LIN {X 0,Y 490.81,Z 849.095,A -85,B 0,C 180,E1 6346.765,E2 6346.765} C_VEL
LIN {X 0,Y 502.24,Z 869.127,A -85,B 0,C 180,E1 6348.343,E2 6348.343} C_VEL
LIN {X 0,Y 506.135,Z 880.489,A -85,B 0,C 180,E1 6348.939,E2 6348.939} C_VEL
LIN {X 0,Y 506.48,Z 902.56,A -85,B 0,C 180,E1 6349.502,E2 6349.502} C_VEL
LIN {X 0,Y 504.044,Z 942.331,A -85,B 0,C 180,E1 6350.762,E2 6350.762} C_VEL
LIN {X 0,Y 500.696,Z 981.834,A -85,B 0,C 180,E1 6352.694,E2 6352.694} C_VEL
LIN {X 0,Y 496.377,Z 1020.467,A -85,B 0,C 180,E1 6355.354,E2 6355.354} C_VEL
LIN {X 0,Y 491.967,Z 1057.531,A -85,B 0,C 180,E1 6358.816,E2 6358.816} C_VEL
LIN {X 0,Y 488.046,Z 1090.045,A -85,B 0,C 180,E1 6362.822,E2 6362.822} C_VEL
LIN {X 0,Y 484.836,Z 1118.607,A -85,B 0,C 180,E1 6367.439,E2 6367.439} C_VEL
LIN {X 0,Y 482.893,Z 1141.028,A -85,B 0,C 180,E1 6372.278,E2 6372.278} C_VEL
LIN {X 0,Y 481.875,Z 1157.894,A -85,B 0,C 180,E1 6377.338,E2 6377.338} C_VEL
LIN {X 0,Y 481.493,Z 1167.965,A -85,B 0,C 180,E1 6381.893,E2 6381.893} C_VEL
LIN {X 0,Y 481.381,Z 1173.637,A -85,B 0,C 180,E1 6386.406,E2 6386.406} C_VEL
LIN {X 0,Y 481.589,Z 1174.659,A -85,B 0,C 180,E1 6391.796,E2 6391.796} C_VEL
LIN {X 0,Y 481.47,Z 1169.517,A -85,B 0,C 180,E1 6397.202,E2 6397.202} C_VEL
LIN {X 0,Y 481.863,Z 1159.093,A -85,B 0,C 180,E1 6402.204,E2 6402.204} C_VEL
LIN {X 0,Y 482.758,Z 1143.624,A -85,B 0,C 180,E1 6407.031,E2 6407.031} C_VEL
LIN {X 0,Y 484.428,Z 1123.467,A -85,B 0,C 180,E1 6411.609,E2 6411.609} C_VEL
LIN {X 0,Y 487.13,Z 1097.644,A -85,B 0,C 180,E1 6416.062,E2 6416.062} C_VEL
LIN {X 0,Y 490.74,Z 1067.209,A -85,B 0,C 180,E1 6420.099,E2 6420.099} C_VEL
LIN {X 0,Y 494.961,Z 1032.68,A -85,B 0,C 180,E1 6423.613,E2 6423.613} C_VEL
LIN {X 0,Y 499.305,Z 993.913,A -85,B 0,C 180,E1 6426.573,E2 6426.573} C_VEL
LIN {X 0,Y 503.244,Z 952.671,A -85,B 0,C 180,E1 6428.803,E2 6428.803} C_VEL
LIN {X 0,Y 506.177,Z 910.447,A -85,B 0,C 180,E1 6430.301,E2 6430.301} C_VEL
LIN {X 0,Y 506.494,Z 891.83,A -85,B 0,C 180,E1 6430.779,E2 6430.779} C_VEL
LIN {X 0,Y 482.863,Z 849.068,A -85,B 0,C 180,E1 6434.121,E2 6434.121} C_VEL
LIN {X 0,Y 480.518,Z 843.44,A -85,B 0,C 180,E1 6434.593,E2 6434.593} C_VEL
LIN {X 0,Y 480.5,Z 843.44,A -85,B 0,C 180,E1 6441.091,E2 6441.091} C_VEL
LIN {X 0,Y 480.506,Z 843.44,A -85,B 0,C 180,E1 6447.733,E2 6447.733} C_VEL
LIN {X 0,Y 480.645,Z 843.44,A -85,B 0,C 180,E1 6453.927,E2 6453.927} C_VEL
LIN {X 0,Y 480.883,Z 843.44,A -85,B 0,C 180,E1 6460.289,E2 6460.289} C_VEL
LIN {X 0,Y 480.75,Z 843.44,A -85,B 0,C 180,E1 6466.669,E2 6466.669} C_VEL
LIN {X 0,Y 481.151,Z 843.44,A -85,B 0,C 180,E1 6472.793,E2 6472.793} C_VEL
LIN {X 0,Y 481.429,Z 843.44,A -85,B 0,C 180,E1 6478.204,E2 6478.204} C_VEL
LIN {X 0,Y 481.304,Z 843.44,A -85,B 0,C 180,E1 6483.595,E2 6483.595} C_VEL
LIN {X 0,Y 481.1,Z 843.44,A -85,B 0,C 180,E1 6489.022,E2 6489.022} C_VEL
LIN {X 0,Y 480.975,Z 843.44,A -85,B 0,C 180,E1 6494.535,E2 6494.535} C_VEL
LIN {X 0,Y 480.824,Z 843.44,A -85,B 0,C 180,E1 6500.194,E2 6500.194} C_VEL
LIN {X 0,Y 480.641,Z 843.44,A -85,B 0,C 180,E1 6506.073,E2 6506.073} C_VEL
LIN {X 0,Y 480.662,Z 843.44,A -85,B 0,C 180,E1 6512.255,E2 6512.255} C_VEL
LIN {X 0,Y 480.609,Z 843.44,A -85,B 0,C 180,E1 6518.284,E2 6518.284} C_VEL
LIN {X 0,Y 480.431,Z 843.44,A -85,B 0,C 180,E1 6524.667,E2 6524.667} C_VEL
LIN {X 0,Y 480.436,Z 843.44,A -85,B 0,C 180,E1 6525.947,E2 6525.947} C_VEL
LIN {X 0,Y 482.833,Z 849.122,A -85,B 0,C 180,E1 6526.359,E2 6526.359} C_VEL
LIN {X 0,Y 501.939,Z 884.383,A -85,B 0,C 180,E1 6529.34,E2 6529.34} C_VEL
LIN {X 0,Y 505.498,Z 893.524,A -85,B 0,C 180,E1 6530.018,E2 6530.018} C_VEL
LIN {X 0,Y 502.302,Z 933.778,A -85,B 0,C 180,E1 6531.656,E2 6531.656} C_VEL
LIN {X 0,Y 498.363,Z 973.134,A -85,B 0,C 180,E1 6534.015,E2 6534.015} C_VEL
LIN {X 0,Y 494.317,Z 1008.152,A -85,B 0,C 180,E1 6536.843,E2 6536.843} C_VEL
LIN {X 0,Y 490.106,Z 1042.495,A -85,B 0,C 180,E1 6540.486,E2 6540.486} C_VEL
LIN {X 0,Y 486.694,Z 1071.747,A -85,B 0,C 180,E1 6544.52,E2 6544.52} C_VEL
LIN {X 0,Y 484.044,Z 1097.342,A -85,B 0,C 180,E1 6549.119,E2 6549.119} C_VEL
LIN {X 0,Y 482.463,Z 1118.01,A -85,B 0,C 180,E1 6554.117,E2 6554.117} C_VEL
LIN {X 0,Y 481.715,Z 1132.635,A -85,B 0,C 180,E1 6559.166,E2 6559.166} C_VEL
LIN {X 0,Y 481.4,Z 1140.792,A -85,B 0,C 180,E1 6563.701,E2 6563.701} C_VEL
LIN {X 0,Y 481.322,Z 1144.674,A -85,B 0,C 180,E1 6568.203,E2 6568.203} C_VEL
LIN {X 0,Y 481.49,Z 1144.64,A -85,B 0,C 180,E1 6571.796,E2 6571.796} C_VEL
LIN {X 0,Y 481.469,Z 1140.671,A -85,B 0,C 180,E1 6576.298,E2 6576.298} C_VEL
LIN {X 0,Y 481.632,Z 1132.416,A -85,B 0,C 180,E1 6580.835,E2 6580.835} C_VEL
LIN {X 0,Y 482.44,Z 1117.714,A -85,B 0,C 180,E1 6585.884,E2 6585.884} C_VEL
LIN {X 0,Y 484.138,Z 1096.755,A -85,B 0,C 180,E1 6590.915,E2 6590.915} C_VEL
LIN {X 0,Y 486.895,Z 1069.683,A -85,B 0,C 180,E1 6595.715,E2 6595.715} C_VEL
LIN {X 0,Y 490.689,Z 1038.025,A -85,B 0,C 180,E1 6599.958,E2 6599.958} C_VEL
LIN {X 0,Y 494.889,Z 1003.334,A -85,B 0,C 180,E1 6603.511,E2 6603.511} C_VEL
LIN {X 0,Y 499.22,Z 964.699,A -85,B 0,C 180,E1 6606.479,E2 6606.479} C_VEL
LIN {X 0,Y 503.328,Z 922.495,A -85,B 0,C 180,E1 6608.788,E2 6608.788} C_VEL
LIN {X 0,Y 505.245,Z 892.288,A -85,B 0,C 180,E1 6609.96,E2 6609.96} C_VEL
LIN {X 0,Y 488.399,Z 858.95,A -85,B 0,C 180,E1 6612.709,E2 6612.709} C_VEL
LIN {X 0,Y 480.532,Z 844.571,A -85,B 0,C 180,E1 6613.908,E2 6613.908} C_VEL
LIN {X 0,Y 480.456,Z 843.44,A -85,B 0,C 180,E1 6614.045,E2 6614.045} C_VEL
LIN {X 0,Y 480.491,Z 843.44,A -85,B 0,C 180,E1 6621.091,E2 6621.091} C_VEL
LIN {X 0,Y 480.488,Z 843.44,A -85,B 0,C 180,E1 6627.732,E2 6627.732} C_VEL
LIN {X 0,Y 480.629,Z 843.44,A -85,B 0,C 180,E1 6633.926,E2 6633.926} C_VEL
LIN {X 0,Y 480.878,Z 843.44,A -85,B 0,C 180,E1 6640.29,E2 6640.29} C_VEL
LIN {X 0,Y 481.024,Z 843.44,A -85,B 0,C 180,E1 6646.531,E2 6646.531} C_VEL
LIN {X 0,Y 481.094,Z 843.44,A -85,B 0,C 180,E1 6652.793,E2 6652.793} C_VEL
LIN {X 0,Y 481.187,Z 843.44,A -85,B 0,C 180,E1 6658.203,E2 6658.203} C_VEL
LIN {X 0,Y 481.204,Z 843.44,A -85,B 0,C 180,E1 6663.596,E2 6663.596} C_VEL
LIN {X 0,Y 481.035,Z 843.44,A -85,B 0,C 180,E1 6669.024,E2 6669.024} C_VEL
LIN {X 0,Y 480.909,Z 843.44,A -85,B 0,C 180,E1 6674.538,E2 6674.538} C_VEL
LIN {X 0,Y 480.779,Z 843.44,A -85,B 0,C 180,E1 6680.197,E2 6680.197} C_VEL
LIN {X 0,Y 480.656,Z 843.44,A -85,B 0,C 180,E1 6686.073,E2 6686.073} C_VEL
LIN {X 0,Y 480.496,Z 843.44,A -85,B 0,C 180,E1 6692.267,E2 6692.267} C_VEL
LIN {X 0,Y 480.499,Z 843.44,A -85,B 0,C 180,E1 6698.909,E2 6698.909} C_VEL
LIN {X 0,Y 480.502,Z 843.44,A -85,B 0,C 180,E1 6705.471,E2 6705.471} C_VEL
LIN {X 0,Y 483.148,Z 849.333,A -85,B 0,C 180,E1 6705.917,E2 6705.917} C_VEL
LIN {X 0,Y 506.915,Z 892.718,A -85,B 0,C 180,E1 6709.28,E2 6709.28} C_VEL
LIN {X 0,Y 506.48,Z 902.56,A -85,B 0,C 180,E1 6709.502,E2 6709.502} C_VEL
LIN {X 0,Y 502.352,Z 919.588,A -85,B 0,C 180,E1 6709.661,E2 6709.661} C_VEL
LIN {X 0,Y 498.468,Z 934.281,A -85,B 0,C 180,E1 6709.883,E2 6709.883} C_VEL
LIN {X 0,Y 498.29,Z 936.369,A -85,B 0,C 180,E1 6709.957,E2 6709.957} C_VEL
LIN {X 0,Y 494.743,Z 975.909,A -85,B 0,C 180,E1 6711.804,E2 6711.804} C_VEL
LIN {X 0,Y 490.375,Z 1014.463,A -85,B 0,C 180,E1 6714.342,E2 6714.342} C_VEL
LIN {X 0,Y 486.018,Z 1049.277,A -85,B 0,C 180,E1 6717.446,E2 6717.446} C_VEL
LIN {X 0,Y 481.782,Z 1082.08,A -85,B 0,C 180,E1 6721.279,E2 6721.279} C_VEL
LIN {X 0,Y 478.081,Z 1111.509,A -85,B 0,C 180,E1 6725.775,E2 6725.775} C_VEL
LIN {X 0,Y 475.712,Z 1135.127,A -85,B 0,C 180,E1 6730.545,E2 6730.545} C_VEL
LIN {X 0,Y 474.402,Z 1152.46,A -85,B 0,C 180,E1 6735.258,E2 6735.258} C_VEL
LIN {X 0,Y 473.714,Z 1164.477,A -85,B 0,C 180,E1 6739.91,E2 6739.91} C_VEL
LIN {X 0,Y 473.44,Z 1171.926,A -85,B 0,C 180,E1 6744.513,E2 6744.513} C_VEL
LIN {X 0,Y 473.413,Z 1174.659,A -85,B 0,C 180,E1 6748.174,E2 6748.174} C_VEL
LIN {X 0,Y 473.682,Z 1174.659,A -85,B 0,C 180,E1 6751.826,E2 6751.826} C_VEL
LIN {X 0,Y 473.572,Z 1169.517,A -85,B 0,C 180,E1 6757.323,E2 6757.323} C_VEL
LIN {X 0,Y 473.979,Z 1159.094,A -85,B 0,C 180,E1 6762.41,E2 6762.41} C_VEL
LIN {X 0,Y 474.935,Z 1144.322,A -85,B 0,C 180,E1 6767.128,E2 6767.128} C_VEL
LIN {X 0,Y 476.706,Z 1124.784,A -85,B 0,C 180,E1 6771.708,E2 6771.708} C_VEL
LIN {X 0,Y 479.621,Z 1098.807,A -85,B 0,C 180,E1 6776.318,E2 6776.318} C_VEL
LIN {X 0,Y 483.542,Z 1068.064,A -85,B 0,C 180,E1 6780.488,E2 6780.488} C_VEL
LIN {X 0,Y 488.001,Z 1034.185,A -85,B 0,C 180,E1 6784.012,E2 6784.012} C_VEL
LIN {X 0,Y 492.684,Z 995.005,A -85,B 0,C 180,E1 6787.049,E2 6787.049} C_VEL
LIN {X 0,Y 496.933,Z 953.369,A -85,B 0,C 180,E1 6789.341,E2 6789.341} C_VEL
LIN {X 0,Y 500.158,Z 909.461,A -85,B 0,C 180,E1 6790.91,E2 6790.91} C_VEL
LIN {X 0,Y 500.541,Z 895.064,A -85,B 0,C 180,E1 6791.29,E2 6791.29} C_VEL
LIN {X 0,Y 478.011,Z 854.286,A -85,B 0,C 180,E1 6794.575,E2 6794.575} C_VEL
LIN {X 0,Y 472.761,Z 844.95,A -85,B 0,C 180,E1 6795.397,E2 6795.397} C_VEL
LIN {X 0,Y 472.596,Z 843.44,A -85,B 0,C 180,E1 6795.502,E2 6795.502} C_VEL
LIN {X 0,Y 472.593,Z 843.44,A -85,B 0,C 180,E1 6802.652,E2 6802.652} C_VEL
LIN {X 0,Y 472.6,Z 843.44,A -85,B 0,C 180,E1 6809.555,E2 6809.555} C_VEL
LIN {X 0,Y 472.765,Z 843.44,A -85,B 0,C 180,E1 6815.485,E2 6815.485} C_VEL
LIN {X 0,Y 472.969,Z 843.44,A -85,B 0,C 180,E1 6821.395,E2 6821.395} C_VEL
LIN {X 0,Y 472.911,Z 843.44,A -85,B 0,C 180,E1 6827.094,E2 6827.094} C_VEL
LIN {X 0,Y 473.225,Z 843.44,A -85,B 0,C 180,E1 6832.672,E2 6832.672} C_VEL
LIN {X 0,Y 473.519,Z 843.44,A -85,B 0,C 180,E1 6838.174,E2 6838.174} C_VEL
LIN {X 0,Y 473.391,Z 843.44,A -85,B 0,C 180,E1 6843.655,E2 6843.655} C_VEL
LIN {X 0,Y 473.203,Z 843.44,A -85,B 0,C 180,E1 6849.174,E2 6849.174} C_VEL
LIN {X 0,Y 473.037,Z 843.44,A -85,B 0,C 180,E1 6854.785,E2 6854.785} C_VEL
LIN {X 0,Y 472.876,Z 843.44,A -85,B 0,C 180,E1 6860.549,E2 6860.549} C_VEL
LIN {X 0,Y 472.693,Z 843.44,A -85,B 0,C 180,E1 6866.637,E2 6866.637} C_VEL
LIN {X 0,Y 472.682,Z 843.44,A -85,B 0,C 180,E1 6872.867,E2 6872.867} C_VEL
LIN {X 0,Y 472.683,Z 843.44,A -85,B 0,C 180,E1 6877.339,E2 6877.339} C_VEL
LIN {X 0,Y 472.552,Z 843.44,A -85,B 0,C 180,E1 6884.628,E2 6884.628} C_VEL
LIN {X 0,Y 472.549,Z 844.229,A -85,B 0,C 180,E1 6885.045,E2 6885.045} C_VEL
LIN {X 0,Y 495.143,Z 886.055,A -85,B 0,C 180,E1 6888.712,E2 6888.712} C_VEL
LIN {X 0,Y 499.299,Z 896.741,A -85,B 0,C 180,E1 6889.53,E2 6889.53} C_VEL
LIN {X 0,Y 495.695,Z 938.305,A -85,B 0,C 180,E1 6891.297,E2 6891.297} C_VEL
LIN {X 0,Y 491.015,Z 980.034,A -85,B 0,C 180,E1 6893.942,E2 6893.942} C_VEL
LIN {X 0,Y 486.249,Z 1017.853,A -85,B 0,C 180,E1 6897.254,E2 6897.254} C_VEL
LIN {X 0,Y 481.882,Z 1051.227,A -85,B 0,C 180,E1 6901.116,E2 6901.116} C_VEL
LIN {X 0,Y 478.288,Z 1080.412,A -85,B 0,C 180,E1 6905.537,E2 6905.537} C_VEL
LIN {X 0,Y 475.701,Z 1105.305,A -85,B 0,C 180,E1 6910.544,E2 6910.544} C_VEL
LIN {X 0,Y 474.406,Z 1122.606,A -85,B 0,C 180,E1 6915.258,E2 6915.258} C_VEL
LIN {X 0,Y 473.707,Z 1134.569,A -85,B 0,C 180,E1 6919.909,E2 6919.909} C_VEL
LIN {X 0,Y 473.435,Z 1141.974,A -85,B 0,C 180,E1 6924.513,E2 6924.513} C_VEL
LIN {X 0,Y 473.419,Z 1144.674,A -85,B 0,C 180,E1 6928.173,E2 6928.173} C_VEL
LIN {X 0,Y 473.584,Z 1144.64,A -85,B 0,C 180,E1 6931.826,E2 6931.826} C_VEL
LIN {X 0,Y 473.561,Z 1140.672,A -85,B 0,C 180,E1 6936.403,E2 6936.403} C_VEL
LIN {X 0,Y 473.782,Z 1132.417,A -85,B 0,C 180,E1 6941.017,E2 6941.017} C_VEL
LIN {X 0,Y 474.652,Z 1117.718,A -85,B 0,C 180,E1 6946.151,E2 6946.151} C_VEL
LIN {X 0,Y 476.6,Z 1096.207,A -85,B 0,C 180,E1 6951.379,E2 6951.379} C_VEL
LIN {X 0,Y 479.526,Z 1069.687,A -85,B 0,C 180,E1 6956.14,E2 6956.14} C_VEL
LIN {X 0,Y 483.516,Z 1038.683,A -85,B 0,C 180,E1 6960.369,E2 6960.369} C_VEL
LIN {X 0,Y 488.159,Z 1002.687,A -85,B 0,C 180,E1 6964.098,E2 6964.098} C_VEL
LIN {X 0,Y 492.971,Z 963.451,A -85,B 0,C 180,E1 6967.13,E2 6967.13} C_VEL
LIN {X 0,Y 497.16,Z 922.661,A -85,B 0,C 180,E1 6969.37,E2 6969.37} C_VEL
LIN {X 0,Y 498.998,Z 895.17,A -85,B 0,C 180,E1 6970.471,E2 6970.471} C_VEL
LIN {X 0,Y 481.406,Z 860.163,A -85,B 0,C 180,E1 6973.463,E2 6973.463} C_VEL
LIN {X 0,Y 472.816,Z 845.405,A -85,B 0,C 180,E1 6974.807,E2 6974.807} C_VEL
LIN {X 0,Y 472.587,Z 843.44,A -85,B 0,C 180,E1 6975.035,E2 6975.035} C_VEL
LIN {X 0,Y 472.499,Z 843.44,A -85,B 0,C 180,E1 6980.304,E2 6980.304} C_VEL
LIN {X 0,Y 472.507,Z 843.44,A -85,B 0,C 180,E1 6986.134,E2 6986.134} C_VEL
LIN {X 0,Y 472.623,Z 843.44,A -85,B 0,C 180,E1 6991.386,E2 6991.386} C_VEL
LIN {X 0,Y 472.862,Z 843.44,A -85,B 0,C 180,E1 6997.737,E2 6997.737} C_VEL
LIN {X 0,Y 473.044,Z 843.44,A -85,B 0,C 180,E1 7003.316,E2 7003.316} C_VEL
LIN {X 0,Y 473.132,Z 843.44,A -85,B 0,C 180,E1 7008.968,E2 7008.968} C_VEL
LIN {X 0,Y 473.262,Z 843.44,A -85,B 0,C 180,E1 7014.511,E2 7014.511} C_VEL
LIN {X 0,Y 473.445,Z 843.44,A -85,B 0,C 180,E1 7020,E2 7020} C_VEL
LIN {X 0,Y 473.289,Z 843.44,A -85,B 0,C 180,E1 7025.489,E2 7025.489} C_VEL
LIN {X 0,Y 473.066,Z 843.44,A -85,B 0,C 180,E1 7031.034,E2 7031.034} C_VEL
LIN {X 0,Y 472.903,Z 843.44,A -85,B 0,C 180,E1 7036.807,E2 7036.807} C_VEL
LIN {X 0,Y 472.811,Z 843.44,A -85,B 0,C 180,E1 7042.518,E2 7042.518} C_VEL
LIN {X 0,Y 472.649,Z 843.44,A -85,B 0,C 180,E1 7048.613,E2 7048.613} C_VEL
LIN {X 0,Y 472.566,Z 843.44,A -85,B 0,C 180,E1 7055.083,E2 7055.083} C_VEL
LIN {X 0,Y 472.502,Z 843.44,A -85,B 0,C 180,E1 7059.961,E2 7059.961} C_VEL
LIN {X 0,Y 472.615,Z 843.593,A -85,B 0,C 180,E1 7064.558,E2 7064.558} C_VEL
LIN {X 0,Y 475.247,Z 849.335,A -85,B 0,C 180,E1 7064.996,E2 7064.996} C_VEL
LIN {X 0,Y 500.023,Z 893.875,A -85,B 0,C 180,E1 7068.63,E2 7068.63} C_VEL
LIN {X 0,Y 500.54,Z 900.795,A -85,B 0,C 180,E1 7068.876,E2 7068.876} C_VEL
LIN {X 0,Y 498.29,Z 936.369,A -85,B 0,C 180,E1 7069.957,E2 7069.957} C_VEL
LIN {X 0,Y 493.901,Z 953.037,A -85,B 0,C 180,E1 7070.346,E2 7070.346} C_VEL
LIN {X 0,Y 489.333,Z 967.284,A -85,B 0,C 180,E1 7070.756,E2 7070.756} C_VEL
LIN {X 0,Y 489.027,Z 969.274,A -85,B 0,C 180,E1 7070.857,E2 7070.857} C_VEL
LIN {X 0,Y 484.23,Z 1010.674,A -85,B 0,C 180,E1 7073.506,E2 7073.506} C_VEL
LIN {X 0,Y 479.392,Z 1047.786,A -85,B 0,C 180,E1 7076.765,E2 7076.765} C_VEL
LIN {X 0,Y 474.575,Z 1082.079,A -85,B 0,C 180,E1 7080.801,E2 7080.801} C_VEL
LIN {X 0,Y 470.648,Z 1111.509,A -85,B 0,C 180,E1 7085.367,E2 7085.367} C_VEL
LIN {X 0,Y 468.039,Z 1135.128,A -85,B 0,C 180,E1 7090.213,E2 7090.213} C_VEL
LIN {X 0,Y 466.586,Z 1152.46,A -85,B 0,C 180,E1 7095.005,E2 7095.005} C_VEL
LIN {X 0,Y 465.851,Z 1164.477,A -85,B 0,C 180,E1 7099.738,E2 7099.738} C_VEL
LIN {X 0,Y 465.554,Z 1171.926,A -85,B 0,C 180,E1 7104.42,E2 7104.42} C_VEL
LIN {X 0,Y 465.526,Z 1174.659,A -85,B 0,C 180,E1 7108.143,E2 7108.143} C_VEL
LIN {X 0,Y 465.796,Z 1174.659,A -85,B 0,C 180,E1 7111.857,E2 7111.857} C_VEL
LIN {X 0,Y 465.677,Z 1169.517,A -85,B 0,C 180,E1 7117.448,E2 7117.448} C_VEL
LIN {X 0,Y 466.106,Z 1159.094,A -85,B 0,C 180,E1 7122.623,E2 7122.623} C_VEL
LIN {X 0,Y 467.143,Z 1144.321,A -85,B 0,C 180,E1 7127.423,E2 7127.423} C_VEL
LIN {X 0,Y 469.17,Z 1124.095,A -85,B 0,C 180,E1 7132.217,E2 7132.217} C_VEL
LIN {X 0,Y 472.294,Z 1098.375,A -85,B 0,C 180,E1 7136.828,E2 7136.828} C_VEL
LIN {X 0,Y 476.598,Z 1067.13,A -85,B 0,C 180,E1 7141.099,E2 7141.099} C_VEL
LIN {X 0,Y 481.26,Z 1034.183,A -85,B 0,C 180,E1 7144.543,E2 7144.543} C_VEL
LIN {X 0,Y 486.22,Z 994.7,A -85,B 0,C 180,E1 7147.626,E2 7147.626} C_VEL
LIN {X 0,Y 490.784,Z 952.424,A -85,B 0,C 180,E1 7149.965,E2 7149.965} C_VEL
LIN {X 0,Y 494.19,Z 909.163,A -85,B 0,C 180,E1 7151.512,E2 7151.512} C_VEL
LIN {X 0,Y 494.178,Z 897.528,A -85,B 0,C 180,E1 7151.859,E2 7151.859} C_VEL
LIN {X 0,Y 473.078,Z 859.171,A -85,B 0,C 180,E1 7155.059,E2 7155.059} C_VEL
LIN {X 0,Y 464.805,Z 844.897,A -85,B 0,C 180,E1 7156.392,E2 7156.392} C_VEL
LIN {X 0,Y 464.638,Z 843.44,A -85,B 0,C 180,E1 7156.53,E2 7156.53} C_VEL
LIN {X 0,Y 464.58,Z 843.44,A -85,B 0,C 180,E1 7161.894,E2 7161.894} C_VEL
LIN {X 0,Y 464.576,Z 843.44,A -85,B 0,C 180,E1 7167.621,E2 7167.621} C_VEL
LIN {X 0,Y 464.751,Z 843.44,A -85,B 0,C 180,E1 7172.964,E2 7172.964} C_VEL
LIN {X 0,Y 464.974,Z 843.44,A -85,B 0,C 180,E1 7179.085,E2 7179.085} C_VEL
LIN {X 0,Y 464.919,Z 843.44,A -85,B 0,C 180,E1 7184.951,E2 7184.951} C_VEL
LIN {X 0,Y 465.15,Z 843.44,A -85,B 0,C 180,E1 7190.665,E2 7190.665} C_VEL
LIN {X 0,Y 465.412,Z 843.44,A -85,B 0,C 180,E1 7196.282,E2 7196.282} C_VEL
LIN {X 0,Y 465.417,Z 843.44,A -85,B 0,C 180,E1 7201.858,E2 7201.858} C_VEL
LIN {X 0,Y 465.284,Z 843.44,A -85,B 0,C 180,E1 7207.453,E2 7207.453} C_VEL
LIN {X 0,Y 465.164,Z 843.44,A -85,B 0,C 180,E1 7213.29,E2 7213.29} C_VEL
LIN {X 0,Y 464.947,Z 843.44,A -85,B 0,C 180,E1 7219.743,E2 7219.743} C_VEL
LIN {X 0,Y 464.79,Z 843.44,A -85,B 0,C 180,E1 7224.964,E2 7224.964} C_VEL
LIN {X 0,Y 464.717,Z 843.44,A -85,B 0,C 180,E1 7231.3,E2 7231.3} C_VEL
LIN {X 0,Y 464.772,Z 843.44,A -85,B 0,C 180,E1 7235.76,E2 7235.76} C_VEL
LIN {X 0,Y 464.49,Z 843.44,A -85,B 0,C 180,E1 7241.65,E2 7241.65} C_VEL
LIN {X 0,Y 464.556,Z 843.44,A -85,B 0,C 180,E1 7244.023,E2 7244.023} C_VEL
LIN {X 0,Y 466.904,Z 849,A -85,B 0,C 180,E1 7244.447,E2 7244.447} C_VEL
LIN {X 0,Y 487.218,Z 885.36,A -85,B 0,C 180,E1 7247.847,E2 7247.847} C_VEL
LIN {X 0,Y 493.058,Z 899.433,A -85,B 0,C 180,E1 7249.016,E2 7249.016} C_VEL
LIN {X 0,Y 489.344,Z 940.042,A -85,B 0,C 180,E1 7250.79,E2 7250.79} C_VEL
LIN {X 0,Y 484.438,Z 980.993,A -85,B 0,C 180,E1 7253.435,E2 7253.435} C_VEL
LIN {X 0,Y 479.318,Z 1018.358,A -85,B 0,C 180,E1 7256.78,E2 7256.78} C_VEL
LIN {X 0,Y 474.684,Z 1051.449,A -85,B 0,C 180,E1 7260.67,E2 7260.67} C_VEL
LIN {X 0,Y 470.755,Z 1080.492,A -85,B 0,C 180,E1 7265.135,E2 7265.135} C_VEL
LIN {X 0,Y 468.026,Z 1105.303,A -85,B 0,C 180,E1 7270.212,E2 7270.212} C_VEL
LIN {X 0,Y 466.599,Z 1122.603,A -85,B 0,C 180,E1 7275.005,E2 7275.005} C_VEL
LIN {X 0,Y 465.845,Z 1134.568,A -85,B 0,C 180,E1 7279.737,E2 7279.737} C_VEL
LIN {X 0,Y 465.549,Z 1141.974,A -85,B 0,C 180,E1 7284.419,E2 7284.419} C_VEL
LIN {X 0,Y 465.532,Z 1144.674,A -85,B 0,C 180,E1 7288.142,E2 7288.142} C_VEL
LIN {X 0,Y 465.677,Z 1144.641,A -85,B 0,C 180,E1 7291.857,E2 7291.857} C_VEL
LIN {X 0,Y 465.659,Z 1140.673,A -85,B 0,C 180,E1 7296.512,E2 7296.512} C_VEL
LIN {X 0,Y 465.912,Z 1132.419,A -85,B 0,C 180,E1 7301.205,E2 7301.205} C_VEL
LIN {X 0,Y 466.904,Z 1117.722,A -85,B 0,C 180,E1 7306.427,E2 7306.427} C_VEL
LIN {X 0,Y 468.995,Z 1096.304,A -85,B 0,C 180,E1 7311.723,E2 7311.723} C_VEL
LIN {X 0,Y 472.224,Z 1069.691,A -85,B 0,C 180,E1 7316.575,E2 7316.575} C_VEL
LIN {X 0,Y 476.47,Z 1038.416,A -85,B 0,C 180,E1 7320.901,E2 7320.901} C_VEL
LIN {X 0,Y 481.604,Z 1002.008,A -85,B 0,C 180,E1 7324.713,E2 7324.713} C_VEL
LIN {X 0,Y 486.47,Z 964.968,A -85,B 0,C 180,E1 7327.622,E2 7327.622} C_VEL
LIN {X 0,Y 490.962,Z 923.82,A -85,B 0,C 180,E1 7329.922,E2 7329.922} C_VEL
LIN {X 0,Y 492.742,Z 897.967,A -85,B 0,C 180,E1 7330.992,E2 7330.992} C_VEL
LIN {X 0,Y 476.157,Z 864.702,A -85,B 0,C 180,E1 7333.961,E2 7333.961} C_VEL
LIN {X 0,Y 464.703,Z 844.333,A -85,B 0,C 180,E1 7335.843,E2 7335.843} C_VEL
LIN {X 0,Y 464.635,Z 843.44,A -85,B 0,C 180,E1 7336.015,E2 7336.015} C_VEL
LIN {X 0,Y 464.571,Z 843.44,A -85,B 0,C 180,E1 7341.893,E2 7341.893} C_VEL
LIN {X 0,Y 464.587,Z 843.44,A -85,B 0,C 180,E1 7348.69,E2 7348.69} C_VEL
LIN {X 0,Y 464.84,Z 843.44,A -85,B 0,C 180,E1 7355.362,E2 7355.362} C_VEL
LIN {X 0,Y 465.019,Z 843.44,A -85,B 0,C 180,E1 7361.065,E2 7361.065} C_VEL
LIN {X 0,Y 465.223,Z 843.44,A -85,B 0,C 180,E1 7366.877,E2 7366.877} C_VEL
LIN {X 0,Y 465.281,Z 843.44,A -85,B 0,C 180,E1 7372.663,E2 7372.663} C_VEL
LIN {X 0,Y 465.414,Z 843.44,A -85,B 0,C 180,E1 7378.142,E2 7378.142} C_VEL
LIN {X 0,Y 465.408,Z 843.44,A -85,B 0,C 180,E1 7383.718,E2 7383.718} C_VEL
LIN {X 0,Y 465.207,Z 843.44,A -85,B 0,C 180,E1 7389.334,E2 7389.334} C_VEL
LIN {X 0,Y 465.034,Z 843.44,A -85,B 0,C 180,E1 7395.046,E2 7395.046} C_VEL
LIN {X 0,Y 464.927,Z 843.44,A -85,B 0,C 180,E1 7400.917,E2 7400.917} C_VEL
LIN {X 0,Y 464.763,Z 843.44,A -85,B 0,C 180,E1 7407.036,E2 7407.036} C_VEL
LIN {X 0,Y 464.597,Z 843.44,A -85,B 0,C 180,E1 7413.514,E2 7413.514} C_VEL
LIN {X 0,Y 464.56,Z 843.44,A -85,B 0,C 180,E1 7418.778,E2 7418.778} C_VEL
LIN {X 0,Y 464.659,Z 843.44,A -85,B 0,C 180,E1 7423.547,E2 7423.547} C_VEL
LIN {X 0,Y 467.012,Z 849.014,A -85,B 0,C 180,E1 7423.98,E2 7423.98} C_VEL
LIN {X 0,Y 490.584,Z 890.192,A -85,B 0,C 180,E1 7427.578,E2 7427.578} C_VEL
LIN {X 0,Y 494.635,Z 899.5,A -85,B 0,C 180,E1 7428.246,E2 7428.246} C_VEL
LIN {X 0,Y 491.798,Z 941.193,A -85,B 0,C 180,E1 7429.559,E2 7429.559} C_VEL
LIN {X 0,Y 489.027,Z 969.274,A -85,B 0,C 180,E1 7430.857,E2 7430.857} C_VEL
LIN {X 0,Y 484.096,Z 985.37,A -85,B 0,C 180,E1 7431.498,E2 7431.498} C_VEL
LIN {X 0,Y 479.028,Z 1000.787,A -85,B 0,C 180,E1 7432.235,E2 7432.235} C_VEL
LIN {X 0,Y 474.013,Z 1037.238,A -85,B 0,C 180,E1 7435.215,E2 7435.215} C_VEL
LIN {X 0,Y 469.065,Z 1070.93,A -85,B 0,C 180,E1 7438.848,E2 7438.848} C_VEL
LIN {X 0,Y 464.508,Z 1101.716,A -85,B 0,C 180,E1 7443.25,E2 7443.25} C_VEL
LIN {X 0,Y 461.184,Z 1127.652,A -85,B 0,C 180,E1 7448.149,E2 7448.149} C_VEL
LIN {X 0,Y 459.091,Z 1147.866,A -85,B 0,C 180,E1 7453.285,E2 7453.285} C_VEL
LIN {X 0,Y 458.163,Z 1162.527,A -85,B 0,C 180,E1 7458.603,E2 7458.603} C_VEL
LIN {X 0,Y 457.739,Z 1170.731,A -85,B 0,C 180,E1 7463.374,E2 7463.374} C_VEL
LIN {X 0,Y 457.624,Z 1174.659,A -85,B 0,C 180,E1 7468.111,E2 7468.111} C_VEL
LIN {X 0,Y 457.888,Z 1174.659,A -85,B 0,C 180,E1 7471.889,E2 7471.889} C_VEL
LIN {X 0,Y 457.788,Z 1169.517,A -85,B 0,C 180,E1 7477.577,E2 7477.577} C_VEL
LIN {X 0,Y 458.261,Z 1159.095,A -85,B 0,C 180,E1 7482.843,E2 7482.843} C_VEL
LIN {X 0,Y 459.45,Z 1143.629,A -85,B 0,C 180,E1 7487.921,E2 7487.921} C_VEL
LIN {X 0,Y 461.638,Z 1122.954,A -85,B 0,C 180,E1 7492.841,E2 7492.841} C_VEL
LIN {X 0,Y 464.94,Z 1098.373,A -85,B 0,C 180,E1 7497.287,E2 7497.287} C_VEL
LIN {X 0,Y 469.568,Z 1067.129,A -85,B 0,C 180,E1 7501.618,E2 7501.618} C_VEL
LIN {X 0,Y 474.692,Z 1032.675,A -85,B 0,C 180,E1 7505.21,E2 7505.21} C_VEL
LIN {X 0,Y 479.86,Z 994.164,A -85,B 0,C 180,E1 7508.231,E2 7508.231} C_VEL
LIN {X 0,Y 484.567,Z 953.211,A -85,B 0,C 180,E1 7510.525,E2 7510.525} C_VEL
LIN {X 0,Y 488.105,Z 910.919,A -85,B 0,C 180,E1 7512.073,E2 7512.073} C_VEL
LIN {X 0,Y 488.264,Z 900.93,A -85,B 0,C 180,E1 7512.371,E2 7512.371} C_VEL
LIN {X 0,Y 467.447,Z 862.552,A -85,B 0,C 180,E1 7515.676,E2 7515.676} C_VEL
LIN {X 0,Y 456.739,Z 844.473,A -85,B 0,C 180,E1 7517.465,E2 7517.465} C_VEL
LIN {X 0,Y 456.657,Z 843.44,A -85,B 0,C 180,E1 7517.752,E2 7517.752} C_VEL
LIN {X 0,Y 456.642,Z 843.44,A -85,B 0,C 180,E1 7523.501,E2 7523.501} C_VEL
LIN {X 0,Y 456.694,Z 843.44,A -85,B 0,C 180,E1 7530.29,E2 7530.29} C_VEL
LIN {X 0,Y 456.922,Z 843.44,A -85,B 0,C 180,E1 7536.653,E2 7536.653} C_VEL
LIN {X 0,Y 457.125,Z 843.44,A -85,B 0,C 180,E1 7543.2,E2 7543.2} C_VEL
LIN {X 0,Y 457.141,Z 843.44,A -85,B 0,C 180,E1 7548.577,E2 7548.577} C_VEL
LIN {X 0,Y 457.481,Z 843.44,A -85,B 0,C 180,E1 7554.321,E2 7554.321} C_VEL
LIN {X 0,Y 457.599,Z 843.44,A -85,B 0,C 180,E1 7560,E2 7560} C_VEL
LIN {X 0,Y 457.442,Z 843.44,A -85,B 0,C 180,E1 7565.679,E2 7565.679} C_VEL
LIN {X 0,Y 457.273,Z 843.44,A -85,B 0,C 180,E1 7571.419,E2 7571.419} C_VEL
LIN {X 0,Y 457.102,Z 843.44,A -85,B 0,C 180,E1 7577.283,E2 7577.283} C_VEL
LIN {X 0,Y 456.92,Z 843.44,A -85,B 0,C 180,E1 7583.346,E2 7583.346} C_VEL
LIN {X 0,Y 456.778,Z 843.44,A -85,B 0,C 180,E1 7589.704,E2 7589.704} C_VEL
LIN {X 0,Y 456.75,Z 843.44,A -85,B 0,C 180,E1 7596.488,E2 7596.488} C_VEL
LIN {X 0,Y 456.615,Z 843.44,A -85,B 0,C 180,E1 7602.962,E2 7602.962} C_VEL
LIN {X 0,Y 458.975,Z 849.029,A -85,B 0,C 180,E1 7603.42,E2 7603.42} C_VEL
LIN {X 0,Y 479.379,Z 884.837,A -85,B 0,C 180,E1 7606.958,E2 7606.958} C_VEL
LIN {X 0,Y 486.881,Z 902.344,A -85,B 0,C 180,E1 7608.502,E2 7608.502} C_VEL
LIN {X 0,Y 482.849,Z 942.871,A -85,B 0,C 180,E1 7610.334,E2 7610.334} C_VEL
LIN {X 0,Y 477.869,Z 982.233,A -85,B 0,C 180,E1 7612.938,E2 7612.938} C_VEL
LIN {X 0,Y 472.603,Z 1017.954,A -85,B 0,C 180,E1 7616.164,E2 7616.164} C_VEL
LIN {X 0,Y 467.474,Z 1051.84,A -85,B 0,C 180,E1 7620.233,E2 7620.233} C_VEL
LIN {X 0,Y 463.327,Z 1080.608,A -85,B 0,C 180,E1 7624.731,E2 7624.731} C_VEL
LIN {X 0,Y 460.342,Z 1105.301,A -85,B 0,C 180,E1 7629.867,E2 7629.867} C_VEL
LIN {X 0,Y 458.783,Z 1122.599,A -85,B 0,C 180,E1 7634.744,E2 7634.744} C_VEL
LIN {X 0,Y 457.994,Z 1134.566,A -85,B 0,C 180,E1 7639.559,E2 7639.559} C_VEL
LIN {X 0,Y 457.652,Z 1141.973,A -85,B 0,C 180,E1 7644.323,E2 7644.323} C_VEL
LIN {X 0,Y 457.629,Z 1144.673,A -85,B 0,C 180,E1 7648.11,E2 7648.11} C_VEL
LIN {X 0,Y 457.771,Z 1144.641,A -85,B 0,C 180,E1 7651.889,E2 7651.889} C_VEL
LIN {X 0,Y 457.77,Z 1140.674,A -85,B 0,C 180,E1 7656.625,E2 7656.625} C_VEL
LIN {X 0,Y 458.054,Z 1132.42,A -85,B 0,C 180,E1 7661.4,E2 7661.4} C_VEL
LIN {X 0,Y 459.154,Z 1117.725,A -85,B 0,C 180,E1 7666.712,E2 7666.712} C_VEL
LIN {X 0,Y 461.415,Z 1096.339,A -85,B 0,C 180,E1 7672.092,E2 7672.092} C_VEL
LIN {X 0,Y 464.892,Z 1069.694,A -85,B 0,C 180,E1 7677.028,E2 7677.028} C_VEL
LIN {X 0,Y 469.511,Z 1037.913,A -85,B 0,C 180,E1 7681.477,E2 7681.477} C_VEL
LIN {X 0,Y 474.856,Z 1003.05,A -85,B 0,C 180,E1 7685.204,E2 7685.204} C_VEL
LIN {X 0,Y 480.185,Z 965.005,A -85,B 0,C 180,E1 7688.223,E2 7688.223} C_VEL
LIN {X 0,Y 484.934,Z 923.362,A -85,B 0,C 180,E1 7690.562,E2 7690.562} C_VEL
LIN {X 0,Y 486.615,Z 901.239,A -85,B 0,C 180,E1 7691.487,E2 7691.487} C_VEL
LIN {X 0,Y 469.372,Z 866.051,A -85,B 0,C 180,E1 7694.741,E2 7694.741} C_VEL
LIN {X 0,Y 456.863,Z 845.014,A -85,B 0,C 180,E1 7696.86,E2 7696.86} C_VEL
LIN {X 0,Y 456.699,Z 843.44,A -85,B 0,C 180,E1 7697.081,E2 7697.081} C_VEL
LIN {X 0,Y 456.612,Z 843.44,A -85,B 0,C 180,E1 7703.499,E2 7703.499} C_VEL
LIN {X 0,Y 456.682,Z 843.44,A -85,B 0,C 180,E1 7710.289,E2 7710.289} C_VEL
LIN {X 0,Y 456.92,Z 843.44,A -85,B 0,C 180,E1 7716.654,E2 7716.654} C_VEL
LIN {X 0,Y 457.227,Z 843.44,A -85,B 0,C 180,E1 7723.157,E2 7723.157} C_VEL
LIN {X 0,Y 457.297,Z 843.44,A -85,B 0,C 180,E1 7728.581,E2 7728.581} C_VEL
LIN {X 0,Y 457.451,Z 843.44,A -85,B 0,C 180,E1 7734.321,E2 7734.321} C_VEL
LIN {X 0,Y 457.664,Z 843.44,A -85,B 0,C 180,E1 7740,E2 7740} C_VEL
LIN {X 0,Y 457.478,Z 843.44,A -85,B 0,C 180,E1 7745.679,E2 7745.679} C_VEL
LIN {X 0,Y 457.227,Z 843.44,A -85,B 0,C 180,E1 7751.421,E2 7751.421} C_VEL
LIN {X 0,Y 457.057,Z 843.44,A -85,B 0,C 180,E1 7757.286,E2 7757.286} C_VEL
LIN {X 0,Y 456.922,Z 843.44,A -85,B 0,C 180,E1 7763.347,E2 7763.347} C_VEL
LIN {X 0,Y 456.705,Z 843.44,A -85,B 0,C 180,E1 7769.709,E2 7769.709} C_VEL
LIN {X 0,Y 456.638,Z 843.44,A -85,B 0,C 180,E1 7776.499,E2 7776.499} C_VEL
LIN {X 0,Y 456.676,Z 843.44,A -85,B 0,C 180,E1 7782.468,E2 7782.468} C_VEL
LIN {X 0,Y 459.216,Z 849.169,A -85,B 0,C 180,E1 7782.976,E2 7782.976} C_VEL
LIN {X 0,Y 482.09,Z 888.505,A -85,B 0,C 180,E1 7786.619,E2 7786.619} C_VEL
LIN {X 0,Y 488.526,Z 903.007,A -85,B 0,C 180,E1 7787.719,E2 7787.719} C_VEL
LIN {X 0,Y 485.387,Z 943.979,A -85,B 0,C 180,E1 7789.074,E2 7789.074} C_VEL
LIN {X 0,Y 481.234,Z 983.189,A -85,B 0,C 180,E1 7791.073,E2 7791.073} C_VEL
LIN {X 0,Y 479.028,Z 1000.787,A -85,B 0,C 180,E1 7792.235,E2 7792.235} C_VEL
LIN {X 0,Y 473.593,Z 1016.027,A -85,B 0,C 180,E1 7793.087,E2 7793.087} C_VEL
LIN {X 0,Y 468.202,Z 1030.543,A -85,B 0,C 180,E1 7794.043,E2 7794.043} C_VEL
LIN {X 0,Y 462.986,Z 1064.541,A -85,B 0,C 180,E1 7797.582,E2 7797.582} C_VEL
LIN {X 0,Y 458.503,Z 1093.59,A -85,B 0,C 180,E1 7801.496,E2 7801.496} C_VEL
LIN {X 0,Y 454.579,Z 1119.598,A -85,B 0,C 180,E1 7806.057,E2 7806.057} C_VEL
LIN {X 0,Y 451.943,Z 1141.814,A -85,B 0,C 180,E1 7811.243,E2 7811.243} C_VEL
LIN {X 0,Y 450.526,Z 1157.892,A -85,B 0,C 180,E1 7816.44,E2 7816.44} C_VEL
LIN {X 0,Y 449.942,Z 1167.848,A -85,B 0,C 180,E1 7821.247,E2 7821.247} C_VEL
LIN {X 0,Y 449.772,Z 1173.636,A -85,B 0,C 180,E1 7826.153,E2 7826.153} C_VEL
LIN {X 0,Y 449.989,Z 1174.659,A -85,B 0,C 180,E1 7831.922,E2 7831.922} C_VEL
LIN {X 0,Y 449.883,Z 1170.731,A -85,B 0,C 180,E1 7836.742,E2 7836.742} C_VEL
LIN {X 0,Y 450.294,Z 1162.526,A -85,B 0,C 180,E1 7841.6,E2 7841.6} C_VEL
LIN {X 0,Y 451.378,Z 1147.865,A -85,B 0,C 180,E1 7847.009,E2 7847.009} C_VEL
LIN {X 0,Y 453.736,Z 1126.542,A -85,B 0,C 180,E1 7852.486,E2 7852.486} C_VEL
LIN {X 0,Y 457.411,Z 1099.966,A -85,B 0,C 180,E1 7857.508,E2 7857.508} C_VEL
LIN {X 0,Y 462.274,Z 1068.723,A -85,B 0,C 180,E1 7861.93,E2 7861.93} C_VEL
LIN {X 0,Y 467.936,Z 1032.75,A -85,B 0,C 180,E1 7865.757,E2 7865.757} C_VEL
LIN {X 0,Y 473.533,Z 993.858,A -85,B 0,C 180,E1 7868.837,E2 7868.837} C_VEL
LIN {X 0,Y 478.492,Z 952.981,A -85,B 0,C 180,E1 7871.146,E2 7871.146} C_VEL
LIN {X 0,Y 482.242,Z 910.621,A -85,B 0,C 180,E1 7872.705,E2 7872.705} C_VEL
LIN {X 0,Y 482.074,Z 903.598,A -85,B 0,C 180,E1 7872.953,E2 7872.953} C_VEL
LIN {X 0,Y 461.728,Z 865.886,A -85,B 0,C 180,E1 7876.328,E2 7876.328} C_VEL
LIN {X 0,Y 448.857,Z 844.694,A -85,B 0,C 180,E1 7878.559,E2 7878.559} C_VEL
LIN {X 0,Y 448.736,Z 843.44,A -85,B 0,C 180,E1 7878.812,E2 7878.812} C_VEL
LIN {X 0,Y 448.692,Z 843.44,A -85,B 0,C 180,E1 7885.13,E2 7885.13} C_VEL
LIN {X 0,Y 448.82,Z 843.44,A -85,B 0,C 180,E1 7891.921,E2 7891.921} C_VEL
LIN {X 0,Y 449.075,Z 843.44,A -85,B 0,C 180,E1 7898.308,E2 7898.308} C_VEL
LIN {X 0,Y 449.108,Z 843.44,A -85,B 0,C 180,E1 7904.407,E2 7904.407} C_VEL
LIN {X 0,Y 449.311,Z 843.44,A -85,B 0,C 180,E1 7910.333,E2 7910.333} C_VEL
LIN {X 0,Y 449.594,Z 843.44,A -85,B 0,C 180,E1 7916.151,E2 7916.151} C_VEL
LIN {X 0,Y 449.63,Z 843.44,A -85,B 0,C 180,E1 7921.923,E2 7921.923} C_VEL
LIN {X 0,Y 449.465,Z 843.44,A -85,B 0,C 180,E1 7927.717,E2 7927.717} C_VEL
LIN {X 0,Y 449.352,Z 843.44,A -85,B 0,C 180,E1 7933.595,E2 7933.595} C_VEL
LIN {X 0,Y 449.088,Z 843.44,A -85,B 0,C 180,E1 7939.805,E2 7939.805} C_VEL
LIN {X 0,Y 448.92,Z 843.44,A -85,B 0,C 180,E1 7945.91,E2 7945.91} C_VEL
LIN {X 0,Y 448.823,Z 843.44,A -85,B 0,C 180,E1 7952.802,E2 7952.802} C_VEL
LIN {X 0,Y 448.76,Z 843.44,A -85,B 0,C 180,E1 7959.339,E2 7959.339} C_VEL
LIN {X 0,Y 448.7,Z 844.129,A -85,B 0,C 180,E1 7961.888,E2 7961.888} C_VEL
LIN {X 0,Y 451.423,Z 849.402,A -85,B 0,C 180,E1 7962.398,E2 7962.398} C_VEL
LIN {X 0,Y 471.874,Z 885.055,A -85,B 0,C 180,E1 7966.096,E2 7966.096} C_VEL
LIN {X 0,Y 480.735,Z 905.172,A -85,B 0,C 180,E1 7967.969,E2 7967.969} C_VEL
LIN {X 0,Y 476.503,Z 945.054,A -85,B 0,C 180,E1 7969.831,E2 7969.831} C_VEL
LIN {X 0,Y 471.402,Z 982.963,A -85,B 0,C 180,E1 7972.384,E2 7972.384} C_VEL
LIN {X 0,Y 465.784,Z 1018.77,A -85,B 0,C 180,E1 7975.664,E2 7975.664} C_VEL
LIN {X 0,Y 460.338,Z 1052.006,A -85,B 0,C 180,E1 7979.735,E2 7979.735} C_VEL
LIN {X 0,Y 455.736,Z 1081.729,A -85,B 0,C 180,E1 7984.504,E2 7984.504} C_VEL
LIN {X 0,Y 452.755,Z 1104.408,A -85,B 0,C 180,E1 7989.284,E2 7989.284} C_VEL
LIN {X 0,Y 450.975,Z 1122.596,A -85,B 0,C 180,E1 7994.473,E2 7994.473} C_VEL
LIN {X 0,Y 450.124,Z 1134.564,A -85,B 0,C 180,E1 7999.375,E2 7999.375} C_VEL
LIN {X 0,Y 449.775,Z 1141.972,A -85,B 0,C 180,E1 8004.223,E2 8004.223} C_VEL
LIN {X 0,Y 449.756,Z 1144.673,A -85,B 0,C 180,E1 8008.077,E2 8008.077} C_VEL
LIN {X 0,Y 449.883,Z 1144.641,A -85,B 0,C 180,E1 8011.922,E2 8011.922} C_VEL
LIN {X 0,Y 449.865,Z 1140.675,A -85,B 0,C 180,E1 8016.742,E2 8016.742} C_VEL
LIN {X 0,Y 450.2,Z 1132.422,A -85,B 0,C 180,E1 8021.602,E2 8021.602} C_VEL
LIN {X 0,Y 451.397,Z 1117.729,A -85,B 0,C 180,E1 8027.008,E2 8027.008} C_VEL
LIN {X 0,Y 453.838,Z 1096.342,A -85,B 0,C 180,E1 8032.481,E2 8032.481} C_VEL
LIN {X 0,Y 457.536,Z 1069.698,A -85,B 0,C 180,E1 8037.499,E2 8037.499} C_VEL
LIN {X 0,Y 462.567,Z 1038.345,A -85,B 0,C 180,E1 8041.989,E2 8041.989} C_VEL
LIN {X 0,Y 468.258,Z 1003.458,A -85,B 0,C 180,E1 8045.766,E2 8045.766} C_VEL
LIN {X 0,Y 473.945,Z 965.317,A -85,B 0,C 180,E1 8048.82,E2 8048.82} C_VEL
LIN {X 0,Y 478.858,Z 924.309,A -85,B 0,C 180,E1 8051.153,E2 8051.153} C_VEL
LIN {X 0,Y 480.355,Z 904.145,A -85,B 0,C 180,E1 8052.031,E2 8052.031} C_VEL
LIN {X 0,Y 464.35,Z 870.936,A -85,B 0,C 180,E1 8055.221,E2 8055.221} C_VEL
LIN {X 0,Y 448.877,Z 845.028,A -85,B 0,C 180,E1 8057.97,E2 8057.97} C_VEL
LIN {X 0,Y 448.736,Z 843.44,A -85,B 0,C 180,E1 8058.171,E2 8058.171} C_VEL
LIN {X 0,Y 448.667,Z 843.44,A -85,B 0,C 180,E1 8065.128,E2 8065.128} C_VEL
LIN {X 0,Y 448.811,Z 843.44,A -85,B 0,C 180,E1 8071.921,E2 8071.921} C_VEL
LIN {X 0,Y 449.069,Z 843.44,A -85,B 0,C 180,E1 8078.308,E2 8078.308} C_VEL
LIN {X 0,Y 449.345,Z 843.44,A -85,B 0,C 180,E1 8084.416,E2 8084.416} C_VEL
LIN {X 0,Y 449.455,Z 843.44,A -85,B 0,C 180,E1 8090.336,E2 8090.336} C_VEL
LIN {X 0,Y 449.663,Z 843.44,A -85,B 0,C 180,E1 8096.152,E2 8096.152} C_VEL
LIN {X 0,Y 449.821,Z 843.44,A -85,B 0,C 180,E1 8101.923,E2 8101.923} C_VEL
LIN {X 0,Y 449.482,Z 843.44,A -85,B 0,C 180,E1 8107.717,E2 8107.717} C_VEL
LIN {X 0,Y 449.27,Z 843.44,A -85,B 0,C 180,E1 8113.598,E2 8113.598} C_VEL
LIN {X 0,Y 449.058,Z 843.44,A -85,B 0,C 180,E1 8119.795,E2 8119.795} C_VEL
LIN {X 0,Y 448.928,Z 843.44,A -85,B 0,C 180,E1 8125.91,E2 8125.91} C_VEL
LIN {X 0,Y 448.689,Z 843.44,A -85,B 0,C 180,E1 8132.777,E2 8132.777} C_VEL
LIN {X 0,Y 448.736,Z 843.44,A -85,B 0,C 180,E1 8139.336,E2 8139.336} C_VEL
LIN {X 0,Y 448.745,Z 843.459,A -85,B 0,C 180,E1 8141.401,E2 8141.401} C_VEL
LIN {X 0,Y 450.974,Z 848.883,A -85,B 0,C 180,E1 8141.845,E2 8141.845} C_VEL
LIN {X 0,Y 471.281,Z 882.405,A -85,B 0,C 180,E1 8145.228,E2 8145.228} C_VEL
LIN {X 0,Y 482.537,Z 904.502,A -85,B 0,C 180,E1 8147.125,E2 8147.125} C_VEL
LIN {X 0,Y 479.141,Z 945.822,A -85,B 0,C 180,E1 8148.538,E2 8148.538} C_VEL
LIN {X 0,Y 474.798,Z 984.039,A -85,B 0,C 180,E1 8150.532,E2 8150.532} C_VEL
LIN {X 0,Y 469.372,Z 1022.603,A -85,B 0,C 180,E1 8153.338,E2 8153.338} C_VEL
LIN {X 0,Y 468.202,Z 1030.543,A -85,B 0,C 180,E1 8154.043,E2 8154.043} C_VEL
LIN {X 0,Y 462.733,Z 1044.762,A -85,B 0,C 180,E1 8155.117,E2 8155.117} C_VEL
LIN {X 0,Y 457.016,Z 1058.276,A -85,B 0,C 180,E1 8156.312,E2 8156.312} C_VEL
LIN {X 0,Y 451.551,Z 1091.307,A -85,B 0,C 180,E1 8160.662,E2 8160.662} C_VEL
LIN {X 0,Y 447.293,Z 1118.49,A -85,B 0,C 180,E1 8165.401,E2 8165.401} C_VEL
LIN {X 0,Y 444.315,Z 1140.958,A -85,B 0,C 180,E1 8170.662,E2 8170.662} C_VEL
LIN {X 0,Y 442.71,Z 1157.891,A -85,B 0,C 180,E1 8176.196,E2 8176.196} C_VEL
LIN {X 0,Y 442.049,Z 1168.121,A -85,B 0,C 180,E1 8181.263,E2 8181.263} C_VEL
LIN {X 0,Y 441.864,Z 1173.636,A -85,B 0,C 180,E1 8186.084,E2 8186.084} C_VEL
LIN {X 0,Y 441.912,Z 1175,A -85,B 0,C 180,E1 8190,E2 8190} C_VEL
LIN {X 0,Y 441.932,Z 1173.637,A -85,B 0,C 180,E1 8193.916,E2 8193.916} C_VEL
LIN {X 0,Y 442.063,Z 1167.961,A -85,B 0,C 180,E1 8198.839,E2 8198.839} C_VEL
LIN {X 0,Y 442.658,Z 1157.891,A -85,B 0,C 180,E1 8203.806,E2 8203.806} C_VEL
LIN {X 0,Y 444.263,Z 1140.952,A -85,B 0,C 180,E1 8209.34,E2 8209.34} C_VEL
LIN {X 0,Y 447.234,Z 1118.608,A -85,B 0,C 180,E1 8214.577,E2 8214.577} C_VEL
LIN {X 0,Y 451.494,Z 1091.455,A -85,B 0,C 180,E1 8219.317,E2 8219.317} C_VEL
LIN {X 0,Y 457.049,Z 1058.034,A -85,B 0,C 180,E1 8223.717,E2 8223.717} C_VEL
LIN {X 0,Y 463.276,Z 1019.883,A -85,B 0,C 180,E1 8227.468,E2 8227.468} C_VEL
LIN {X 0,Y 469.062,Z 980.165,A -85,B 0,C 180,E1 8230.322,E2 8230.322} C_VEL
LIN {X 0,Y 473.984,Z 938.09,A -85,B 0,C 180,E1 8232.421,E2 8232.421} C_VEL
LIN {X 0,Y 476.051,Z 906.675,A -85,B 0,C 180,E1 8233.525,E2 8233.525} C_VEL
LIN {X 0,Y 456.97,Z 870.853,A -85,B 0,C 180,E1 8236.84,E2 8236.84} C_VEL
LIN {X 0,Y 440.936,Z 844.516,A -85,B 0,C 180,E1 8239.733,E2 8239.733} C_VEL
LIN {X 0,Y 440.846,Z 843.44,A -85,B 0,C 180,E1 8239.819,E2 8239.819} C_VEL
LIN {X 0,Y 440.743,Z 843.44,A -85,B 0,C 180,E1 8246.785,E2 8246.785} C_VEL
LIN {X 0,Y 440.935,Z 843.44,A -85,B 0,C 180,E1 8253.584,E2 8253.584} C_VEL
LIN {X 0,Y 441.203,Z 843.44,A -85,B 0,C 180,E1 8260,E2 8260} C_VEL
LIN {X 0,Y 441.226,Z 843.44,A -85,B 0,C 180,E1 8266.149,E2 8266.149} C_VEL
LIN {X 0,Y 441.581,Z 843.44,A -85,B 0,C 180,E1 8272.316,E2 8272.316} C_VEL
LIN {X 0,Y 441.91,Z 843.44,A -85,B 0,C 180,E1 8278.043,E2 8278.043} C_VEL
LIN {X 0,Y 441.747,Z 843.44,A -85,B 0,C 180,E1 8283.917,E2 8283.917} C_VEL
LIN {X 0,Y 441.516,Z 843.44,A -85,B 0,C 180,E1 8289.839,E2 8289.839} C_VEL
LIN {X 0,Y 441.31,Z 843.44,A -85,B 0,C 180,E1 8295.875,E2 8295.875} C_VEL
LIN {X 0,Y 441.047,Z 843.44,A -85,B 0,C 180,E1 8302.513,E2 8302.513} C_VEL
LIN {X 0,Y 440.95,Z 843.44,A -85,B 0,C 180,E1 8308.626,E2 8308.626} C_VEL
LIN {X 0,Y 440.897,Z 843.44,A -85,B 0,C 180,E1 8315.578,E2 8315.578} C_VEL
LIN {X 0,Y 440.768,Z 843.46,A -85,B 0,C 180,E1 8320.699,E2 8320.699} C_VEL
LIN {X 0,Y 443.106,Z 849.035,A -85,B 0,C 180,E1 8321.187,E2 8321.187} C_VEL
LIN {X 0,Y 461.618,Z 880.046,A -85,B 0,C 180,E1 8324.652,E2 8324.652} C_VEL
LIN {X 0,Y 474.635,Z 907.581,A -85,B 0,C 180,E1 8327.403,E2 8327.403} C_VEL
LIN {X 0,Y 470.181,Z 947.217,A -85,B 0,C 180,E1 8329.312,E2 8329.312} C_VEL
LIN {X 0,Y 464.776,Z 984.888,A -85,B 0,C 180,E1 8331.911,E2 8331.911} C_VEL
LIN {X 0,Y 459.031,Z 1019.52,A -85,B 0,C 180,E1 8335.144,E2 8335.144} C_VEL
LIN {X 0,Y 453.301,Z 1052.306,A -85,B 0,C 180,E1 8339.214,E2 8339.214} C_VEL
LIN {X 0,Y 448.342,Z 1081.723,A -85,B 0,C 180,E1 8344.052,E2 8344.052} C_VEL
LIN {X 0,Y 445.042,Z 1104.865,A -85,B 0,C 180,E1 8349.029,E2 8349.029} C_VEL
LIN {X 0,Y 443.175,Z 1122.593,A -85,B 0,C 180,E1 8354.193,E2 8354.193} C_VEL
LIN {X 0,Y 442.256,Z 1134.562,A -85,B 0,C 180,E1 8359.183,E2 8359.183} C_VEL
LIN {X 0,Y 441.877,Z 1141.971,A -85,B 0,C 180,E1 8364.12,E2 8364.12} C_VEL
LIN {X 0,Y 441.852,Z 1144.673,A -85,B 0,C 180,E1 8368.043,E2 8368.043} C_VEL
LIN {X 0,Y 441.977,Z 1144.642,A -85,B 0,C 180,E1 8371.956,E2 8371.956} C_VEL
LIN {X 0,Y 441.971,Z 1140.676,A -85,B 0,C 180,E1 8376.863,E2 8376.863} C_VEL
LIN {X 0,Y 442.353,Z 1132.423,A -85,B 0,C 180,E1 8381.811,E2 8381.811} C_VEL
LIN {X 0,Y 443.626,Z 1117.733,A -85,B 0,C 180,E1 8387.315,E2 8387.315} C_VEL
LIN {X 0,Y 446.274,Z 1096.344,A -85,B 0,C 180,E1 8392.883,E2 8392.883} C_VEL
LIN {X 0,Y 450.275,Z 1069.813,A -85,B 0,C 180,E1 8397.981,E2 8397.981} C_VEL
LIN {X 0,Y 455.719,Z 1038.656,A -85,B 0,C 180,E1 8402.528,E2 8402.528} C_VEL
LIN {X 0,Y 461.618,Z 1004.474,A -85,B 0,C 180,E1 8406.287,E2 8406.287} C_VEL
LIN {X 0,Y 467.671,Z 966.142,A -85,B 0,C 180,E1 8409.4,E2 8409.4} C_VEL
LIN {X 0,Y 472.92,Z 924.685,A -85,B 0,C 180,E1 8411.781,E2 8411.781} C_VEL
LIN {X 0,Y 474.32,Z 907.372,A -85,B 0,C 180,E1 8412.553,E2 8412.553} C_VEL
LIN {X 0,Y 457.445,Z 872.083,A -85,B 0,C 180,E1 8416.073,E2 8416.073} C_VEL
LIN {X 0,Y 442.162,Z 847.873,A -85,B 0,C 180,E1 8418.886,E2 8418.886} C_VEL
LIN {X 0,Y 440.803,Z 843.44,A -85,B 0,C 180,E1 8419.304,E2 8419.304} C_VEL
LIN {X 0,Y 440.761,Z 843.44,A -85,B 0,C 180,E1 8425.253,E2 8425.253} C_VEL
LIN {X 0,Y 440.889,Z 843.44,A -85,B 0,C 180,E1 8431.37,E2 8431.37} C_VEL
LIN {X 0,Y 441.097,Z 843.44,A -85,B 0,C 180,E1 8437.896,E2 8437.896} C_VEL
LIN {X 0,Y 441.394,Z 843.44,A -85,B 0,C 180,E1 8444.128,E2 8444.128} C_VEL
LIN {X 0,Y 441.544,Z 843.44,A -85,B 0,C 180,E1 8450.162,E2 8450.162} C_VEL
LIN {X 0,Y 441.75,Z 843.44,A -85,B 0,C 180,E1 8456.083,E2 8456.083} C_VEL
LIN {X 0,Y 441.909,Z 843.44,A -85,B 0,C 180,E1 8461.957,E2 8461.957} C_VEL
LIN {X 0,Y 441.586,Z 843.44,A -85,B 0,C 180,E1 8467.856,E2 8467.856} C_VEL
LIN {X 0,Y 441.332,Z 843.44,A -85,B 0,C 180,E1 8473.848,E2 8473.848} C_VEL
LIN {X 0,Y 441.147,Z 843.44,A -85,B 0,C 180,E1 8480.002,E2 8480.002} C_VEL
LIN {X 0,Y 440.948,Z 843.44,A -85,B 0,C 180,E1 8486.415,E2 8486.415} C_VEL
LIN {X 0,Y 440.74,Z 843.44,A -85,B 0,C 180,E1 8493.216,E2 8493.216} C_VEL
LIN {X 0,Y 440.842,Z 843.44,A -85,B 0,C 180,E1 8500.23,E2 8500.23} C_VEL
LIN {X 0,Y 443.284,Z 849.139,A -85,B 0,C 180,E1 8500.74,E2 8500.74} C_VEL
LIN {X 0,Y 464.032,Z 882.962,A -85,B 0,C 180,E1 8504.357,E2 8504.357} C_VEL
LIN {X 0,Y 476.532,Z 908.211,A -85,B 0,C 180,E1 8506.578,E2 8506.578} C_VEL
LIN {X 0,Y 472.593,Z 951.043,A -85,B 0,C 180,E1 8508.135,E2 8508.135} C_VEL
LIN {X 0,Y 467.599,Z 991.049,A -85,B 0,C 180,E1 8510.378,E2 8510.378} C_VEL
LIN {X 0,Y 461.753,Z 1029.104,A -85,B 0,C 180,E1 8513.343,E2 8513.343} C_VEL
LIN {X 0,Y 457.016,Z 1058.276,A -85,B 0,C 180,E1 8516.312,E2 8516.312} C_VEL
LIN {X 0,Y 451.216,Z 1071.291,A -85,B 0,C 180,E1 8517.624,E2 8517.624} C_VEL
LIN {X 0,Y 445.991,Z 1082.098,A -85,B 0,C 180,E1 8518.838,E2 8518.838} C_VEL
LIN {X 0,Y 445.687,Z 1083.522,A -85,B 0,C 180,E1 8519.044,E2 8519.044} C_VEL
LIN {X 0,Y 440.979,Z 1111.33,A -85,B 0,C 180,E1 8523.586,E2 8523.586} C_VEL
LIN {X 0,Y 437.461,Z 1134.68,A -85,B 0,C 180,E1 8528.643,E2 8528.643} C_VEL
LIN {X 0,Y 435.248,Z 1153.893,A -85,B 0,C 180,E1 8534.414,E2 8534.414} C_VEL
LIN {X 0,Y 434.26,Z 1166.392,A -85,B 0,C 180,E1 8539.995,E2 8539.995} C_VEL
LIN {X 0,Y 433.986,Z 1171.926,A -85,B 0,C 180,E1 8544.013,E2 8544.013} C_VEL
LIN {X 0,Y 433.943,Z 1174.659,A -85,B 0,C 180,E1 8548.007,E2 8548.007} C_VEL
LIN {X 0,Y 434.171,Z 1174.659,A -85,B 0,C 180,E1 8551.992,E2 8551.992} C_VEL
LIN {X 0,Y 434.115,Z 1170.731,A -85,B 0,C 180,E1 8556.988,E2 8556.988} C_VEL
LIN {X 0,Y 434.551,Z 1162.525,A -85,B 0,C 180,E1 8562.026,E2 8562.026} C_VEL
LIN {X 0,Y 435.803,Z 1148.011,A -85,B 0,C 180,E1 8567.588,E2 8567.588} C_VEL
LIN {X 0,Y 438.402,Z 1127.646,A -85,B 0,C 180,E1 8573.05,E2 8573.05} C_VEL
LIN {X 0,Y 442.204,Z 1103.327,A -85,B 0,C 180,E1 8577.848,E2 8577.848} C_VEL
LIN {X 0,Y 447.429,Z 1073.102,A -85,B 0,C 180,E1 8582.394,E2 8582.394} C_VEL
LIN {X 0,Y 453.25,Z 1040.375,A -85,B 0,C 180,E1 8586.158,E2 8586.158} C_VEL
LIN {X 0,Y 459.257,Z 1003.793,A -85,B 0,C 180,E1 8589.353,E2 8589.353} C_VEL
LIN {X 0,Y 465.039,Z 963.525,A -85,B 0,C 180,E1 8591.894,E2 8591.894} C_VEL
LIN {X 0,Y 469.671,Z 920.974,A -85,B 0,C 180,E1 8593.695,E2 8593.695} C_VEL
LIN {X 0,Y 470.021,Z 909.523,A -85,B 0,C 180,E1 8594.115,E2 8594.115} C_VEL
LIN {X 0,Y 451.597,Z 874.619,A -85,B 0,C 180,E1 8597.479,E2 8597.479} C_VEL
LIN {X 0,Y 434.978,Z 848.756,A -85,B 0,C 180,E1 8600.552,E2 8600.552} C_VEL
LIN {X 0,Y 432.92,Z 843.44,A -85,B 0,C 180,E1 8601.142,E2 8601.142} C_VEL
LIN {X 0,Y 432.806,Z 843.44,A -85,B 0,C 180,E1 8608.468,E2 8608.468} C_VEL
LIN {X 0,Y 433.044,Z 843.44,A -85,B 0,C 180,E1 8615.282,E2 8615.282} C_VEL
LIN {X 0,Y 433.294,Z 843.44,A -85,B 0,C 180,E1 8621.734,E2 8621.734} C_VEL
LIN {X 0,Y 433.355,Z 843.44,A -85,B 0,C 180,E1 8627.941,E2 8627.941} C_VEL
LIN {X 0,Y 433.764,Z 843.44,A -85,B 0,C 180,E1 8634.009,E2 8634.009} C_VEL
LIN {X 0,Y 433.91,Z 843.44,A -85,B 0,C 180,E1 8640,E2 8640} C_VEL
LIN {X 0,Y 433.717,Z 843.44,A -85,B 0,C 180,E1 8645.991,E2 8645.991} C_VEL
LIN {X 0,Y 433.46,Z 843.44,A -85,B 0,C 180,E1 8652.896,E2 8652.896} C_VEL
LIN {X 0,Y 433.285,Z 843.44,A -85,B 0,C 180,E1 8658.266,E2 8658.266} C_VEL
LIN {X 0,Y 433.018,Z 843.44,A -85,B 0,C 180,E1 8665.032,E2 8665.032} C_VEL
LIN {X 0,Y 432.958,Z 843.44,A -85,B 0,C 180,E1 8671.519,E2 8671.519} C_VEL
LIN {X 0,Y 432.89,Z 843.44,A -85,B 0,C 180,E1 8676.701,E2 8676.701} C_VEL
LIN {X 0,Y 432.846,Z 844.153,A -85,B 0,C 180,E1 8679.471,E2 8679.471} C_VEL
LIN {X 0,Y 435.573,Z 849.44,A -85,B 0,C 180,E1 8680.042,E2 8680.042} C_VEL
LIN {X 0,Y 454.61,Z 881.133,A -85,B 0,C 180,E1 8683.777,E2 8683.777} C_VEL
LIN {X 0,Y 468.574,Z 910.776,A -85,B 0,C 180,E1 8686.86,E2 8686.86} C_VEL
LIN {X 0,Y 463.446,Z 953.229,A -85,B 0,C 180,E1 8689.012,E2 8689.012} C_VEL
LIN {X 0,Y 457.086,Z 993.415,A -85,B 0,C 180,E1 8691.972,E2 8691.972} C_VEL
LIN {X 0,Y 450.564,Z 1030.14,A -85,B 0,C 180,E1 8695.731,E2 8695.731} C_VEL
LIN {X 0,Y 444.539,Z 1062.032,A -85,B 0,C 180,E1 8700.098,E2 8700.098} C_VEL
LIN {X 0,Y 439.923,Z 1088.632,A -85,B 0,C 180,E1 8704.932,E2 8704.932} C_VEL
LIN {X 0,Y 436.614,Z 1111.113,A -85,B 0,C 180,E1 8710.307,E2 8710.307} C_VEL
LIN {X 0,Y 434.878,Z 1128.008,A -85,B 0,C 180,E1 8715.942,E2 8715.942} C_VEL
LIN {X 0,Y 434.157,Z 1138.035,A -85,B 0,C 180,E1 8721.001,E2 8721.001} C_VEL
LIN {X 0,Y 433.988,Z 1143.665,A -85,B 0,C 180,E1 8726.012,E2 8726.012} C_VEL
LIN {X 0,Y 434.009,Z 1144.998,A -85,B 0,C 180,E1 8730,E2 8730} C_VEL
LIN {X 0,Y 434.016,Z 1143.604,A -85,B 0,C 180,E1 8733.987,E2 8733.987} C_VEL
LIN {X 0,Y 434.227,Z 1137.896,A -85,B 0,C 180,E1 8738.997,E2 8738.997} C_VEL
LIN {X 0,Y 434.925,Z 1127.773,A -85,B 0,C 180,E1 8744.056,E2 8744.056} C_VEL
LIN {X 0,Y 436.548,Z 1110.791,A -85,B 0,C 180,E1 8749.696,E2 8749.696} C_VEL
LIN {X 0,Y 439.897,Z 1088.213,A -85,B 0,C 180,E1 8755.07,E2 8755.07} C_VEL
LIN {X 0,Y 444.934,Z 1059.911,A -85,B 0,C 180,E1 8760.138,E2 8760.138} C_VEL
LIN {X 0,Y 450.905,Z 1028.357,A -85,B 0,C 180,E1 8764.384,E2 8764.384} C_VEL
LIN {X 0,Y 457.217,Z 993.184,A -85,B 0,C 180,E1 8767.947,E2 8767.947} C_VEL
LIN {X 0,Y 463.271,Z 954.999,A -85,B 0,C 180,E1 8770.781,E2 8770.781} C_VEL
LIN {X 0,Y 468.291,Z 914.19,A -85,B 0,C 180,E1 8772.9,E2 8772.9} C_VEL
LIN {X 0,Y 467.646,Z 909.077,A -85,B 0,C 180,E1 8773.242,E2 8773.242} C_VEL
LIN {X 0,Y 451.768,Z 875.78,A -85,B 0,C 180,E1 8776.704,E2 8776.704} C_VEL
LIN {X 0,Y 434.887,Z 848.759,A -85,B 0,C 180,E1 8779.986,E2 8779.986} C_VEL
LIN {X 0,Y 432.796,Z 843.44,A -85,B 0,C 180,E1 8780.525,E2 8780.525} C_VEL
LIN {X 0,Y 432.824,Z 843.44,A -85,B 0,C 180,E1 8786.798,E2 8786.798} C_VEL
LIN {X 0,Y 433,Z 843.44,A -85,B 0,C 180,E1 8793.062,E2 8793.062} C_VEL
LIN {X 0,Y 433.319,Z 843.44,A -85,B 0,C 180,E1 8800.095,E2 8800.095} C_VEL
LIN {X 0,Y 433.548,Z 843.44,A -85,B 0,C 180,E1 8805.899,E2 8805.899} C_VEL
LIN {X 0,Y 433.611,Z 843.44,A -85,B 0,C 180,E1 8812.647,E2 8812.647} C_VEL
LIN {X 0,Y 433.819,Z 843.44,A -85,B 0,C 180,E1 8818.007,E2 8818.007} C_VEL
LIN {X 0,Y 433.776,Z 843.44,A -85,B 0,C 180,E1 8823.99,E2 8823.99} C_VEL
LIN {X 0,Y 433.537,Z 843.44,A -85,B 0,C 180,E1 8830.022,E2 8830.022} C_VEL
LIN {X 0,Y 433.339,Z 843.44,A -85,B 0,C 180,E1 8836.175,E2 8836.175} C_VEL
LIN {X 0,Y 433.177,Z 843.44,A -85,B 0,C 180,E1 8842.531,E2 8842.531} C_VEL
LIN {X 0,Y 432.89,Z 843.44,A -85,B 0,C 180,E1 8849.37,E2 8849.37} C_VEL
LIN {X 0,Y 432.79,Z 843.44,A -85,B 0,C 180,E1 8856.35,E2 8856.35} C_VEL
LIN {X 0,Y 432.911,Z 843.44,A -85,B 0,C 180,E1 8858.984,E2 8858.984} C_VEL
LIN {X 0,Y 435.16,Z 848.964,A -85,B 0,C 180,E1 8859.49,E2 8859.49} C_VEL
LIN {X 0,Y 454.839,Z 880.219,A -85,B 0,C 180,E1 8863.101,E2 8863.101} C_VEL
LIN {X 0,Y 470.432,Z 910.497,A -85,B 0,C 180,E1 8865.972,E2 8865.972} C_VEL
LIN {X 0,Y 466.306,Z 953.657,A -85,B 0,C 180,E1 8867.613,E2 8867.613} C_VEL
LIN {X 0,Y 460.974,Z 993.374,A -85,B 0,C 180,E1 8869.904,E2 8869.904} C_VEL
LIN {X 0,Y 454.547,Z 1032.947,A -85,B 0,C 180,E1 8873.105,E2 8873.105} C_VEL
LIN {X 0,Y 448.183,Z 1069.375,A -85,B 0,C 180,E1 8877.117,E2 8877.117} C_VEL
LIN {X 0,Y 445.687,Z 1083.522,A -85,B 0,C 180,E1 8879.044,E2 8879.044} C_VEL
LIN {X 0,Y 441.912,Z 1092.379,A -85,B 0,C 180,E1 8880.213,E2 8880.213} C_VEL
LIN {X 0,Y 434.674,Z 1104.883,A -85,B 0,C 180,E1 8881.98,E2 8881.98} C_VEL
LIN {X 0,Y 434.359,Z 1106.178,A -85,B 0,C 180,E1 8882.206,E2 8882.206} C_VEL
LIN {X 0,Y 430.348,Z 1130.803,A -85,B 0,C 180,E1 8887.312,E2 8887.312} C_VEL
LIN {X 0,Y 427.844,Z 1149.321,A -85,B 0,C 180,E1 8892.527,E2 8892.527} C_VEL
LIN {X 0,Y 426.7,Z 1162.525,A -85,B 0,C 180,E1 8897.75,E2 8897.75} C_VEL
LIN {X 0,Y 426.203,Z 1170.222,A -85,B 0,C 180,E1 8902.45,E2 8902.45} C_VEL
LIN {X 0,Y 426.039,Z 1174.659,A -85,B 0,C 180,E1 8907.97,E2 8907.97} C_VEL
LIN {X 0,Y 426.263,Z 1174.659,A -85,B 0,C 180,E1 8912.029,E2 8912.029} C_VEL
LIN {X 0,Y 426.221,Z 1170.201,A -85,B 0,C 180,E1 8917.568,E2 8917.568} C_VEL
LIN {X 0,Y 426.778,Z 1160.922,A -85,B 0,C 180,E1 8922.976,E2 8922.976} C_VEL
LIN {X 0,Y 428.26,Z 1146.177,A -85,B 0,C 180,E1 8928.489,E2 8928.489} C_VEL
LIN {X 0,Y 430.922,Z 1126.752,A -85,B 0,C 180,E1 8933.654,E2 8933.654} C_VEL
LIN {X 0,Y 435.593,Z 1099.265,A -85,B 0,C 180,E1 8939.013,E2 8939.013} C_VEL
LIN {X 0,Y 441.657,Z 1066.978,A -85,B 0,C 180,E1 8943.726,E2 8943.726} C_VEL
LIN {X 0,Y 448.275,Z 1031.484,A -85,B 0,C 180,E1 8947.625,E2 8947.625} C_VEL
LIN {X 0,Y 454.61,Z 994.161,A -85,B 0,C 180,E1 8950.682,E2 8950.682} C_VEL
LIN {X 0,Y 460.413,Z 953.568,A -85,B 0,C 180,E1 8953.046,E2 8953.046} C_VEL
LIN {X 0,Y 464.146,Z 912.916,A -85,B 0,C 180,E1 8954.67,E2 8954.67} C_VEL
LIN {X 0,Y 445.876,Z 877.683,A -85,B 0,C 180,E1 8958.206,E2 8958.206} C_VEL
LIN {X 0,Y 427.378,Z 849.163,A -85,B 0,C 180,E1 8961.786,E2 8961.786} C_VEL
LIN {X 0,Y 424.932,Z 844.193,A -85,B 0,C 180,E1 8962.336,E2 8962.336} C_VEL
LIN {X 0,Y 424.913,Z 843.44,A -85,B 0,C 180,E1 8968.466,E2 8968.466} C_VEL
LIN {X 0,Y 425.111,Z 843.44,A -85,B 0,C 180,E1 8974.789,E2 8974.789} C_VEL
LIN {X 0,Y 425.368,Z 843.44,A -85,B 0,C 180,E1 8981.381,E2 8981.381} C_VEL
LIN {X 0,Y 425.466,Z 843.44,A -85,B 0,C 180,E1 8987.714,E2 8987.714} C_VEL
LIN {X 0,Y 425.841,Z 843.44,A -85,B 0,C 180,E1 8993.898,E2 8993.898} C_VEL
LIN {X 0,Y 426.009,Z 843.44,A -85,B 0,C 180,E1 9000,E2 9000} C_VEL
LIN {X 0,Y 425.798,Z 843.44,A -85,B 0,C 180,E1 9006.103,E2 9006.103} C_VEL
LIN {X 0,Y 425.613,Z 843.44,A -85,B 0,C 180,E1 9012.282,E2 9012.282} C_VEL
LIN {X 0,Y 425.358,Z 843.44,A -85,B 0,C 180,E1 9018.619,E2 9018.619} C_VEL
LIN {X 0,Y 425.117,Z 843.44,A -85,B 0,C 180,E1 9025.21,E2 9025.21} C_VEL
LIN {X 0,Y 425.034,Z 843.44,A -85,B 0,C 180,E1 9032.176,E2 9032.176} C_VEL
LIN {X 0,Y 424.891,Z 843.44,A -85,B 0,C 180,E1 9038.095,E2 9038.095} C_VEL
LIN {X 0,Y 427.227,Z 849.019,A -85,B 0,C 180,E1 9038.668,E2 9038.668} C_VEL
LIN {X 0,Y 443.989,Z 875.538,A -85,B 0,C 180,E1 9042.098,E2 9042.098} C_VEL
LIN {X 0,Y 460.89,Z 909.884,A -85,B 0,C 180,E1 9045.894,E2 9045.894} C_VEL
LIN {X 0,Y 462.288,Z 916.114,A -85,B 0,C 180,E1 9046.407,E2 9046.407} C_VEL
LIN {X 0,Y 457.015,Z 956.519,A -85,B 0,C 180,E1 9048.55,E2 9048.55} C_VEL
LIN {X 0,Y 450.484,Z 995.166,A -85,B 0,C 180,E1 9051.472,E2 9051.472} C_VEL
LIN {X 0,Y 443.66,Z 1031.467,A -85,B 0,C 180,E1 9055.269,E2 9055.269} C_VEL
LIN {X 0,Y 437.466,Z 1062.414,A -85,B 0,C 180,E1 9059.578,E2 9059.578} C_VEL
LIN {X 0,Y 432.368,Z 1089.905,A -85,B 0,C 180,E1 9064.688,E2 9064.688} C_VEL
LIN {X 0,Y 428.688,Z 1112.86,A -85,B 0,C 180,E1 9070.463,E2 9070.463} C_VEL
LIN {X 0,Y 427.049,Z 1128.005,A -85,B 0,C 180,E1 9075.679,E2 9075.679} C_VEL
LIN {X 0,Y 426.28,Z 1138.033,A -85,B 0,C 180,E1 9080.834,E2 9080.834} C_VEL
LIN {X 0,Y 426.078,Z 1143.664,A -85,B 0,C 180,E1 9085.938,E2 9085.938} C_VEL
LIN {X 0,Y 426.108,Z 1144.998,A -85,B 0,C 180,E1 9090,E2 9090} C_VEL
LIN {X 0,Y 426.109,Z 1143.605,A -85,B 0,C 180,E1 9094.061,E2 9094.061} C_VEL
LIN {X 0,Y 426.359,Z 1137.897,A -85,B 0,C 180,E1 9099.164,E2 9099.164} C_VEL
LIN {X 0,Y 427.072,Z 1127.775,A -85,B 0,C 180,E1 9104.32,E2 9104.32} C_VEL
LIN {X 0,Y 428.654,Z 1112.574,A -85,B 0,C 180,E1 9109.538,E2 9109.538} C_VEL
LIN {X 0,Y 432.357,Z 1089.53,A -85,B 0,C 180,E1 9115.312,E2 9115.312} C_VEL
LIN {X 0,Y 437.664,Z 1061.573,A -85,B 0,C 180,E1 9120.466,E2 9120.466} C_VEL
LIN {X 0,Y 444.225,Z 1028.667,A -85,B 0,C 180,E1 9124.976,E2 9124.976} C_VEL
LIN {X 0,Y 450.853,Z 993.763,A -85,B 0,C 180,E1 9128.553,E2 9128.553} C_VEL
LIN {X 0,Y 457.257,Z 955.309,A -85,B 0,C 180,E1 9131.434,E2 9131.434} C_VEL
LIN {X 0,Y 462.345,Z 914.106,A -85,B 0,C 180,E1 9133.612,E2 9133.612} C_VEL
LIN {X 0,Y 447.172,Z 881.206,A -85,B 0,C 180,E1 9137.144,E2 9137.144} C_VEL
LIN {X 0,Y 430.891,Z 854.575,A -85,B 0,C 180,E1 9140.479,E2 9140.479} C_VEL
LIN {X 0,Y 424.963,Z 844.741,A -85,B 0,C 180,E1 9141.732,E2 9141.732} C_VEL
LIN {X 0,Y 424.864,Z 843.44,A -85,B 0,C 180,E1 9141.81,E2 9141.81} C_VEL
LIN {X 0,Y 424.907,Z 843.44,A -85,B 0,C 180,E1 9148.466,E2 9148.466} C_VEL
LIN {X 0,Y 425.103,Z 843.44,A -85,B 0,C 180,E1 9154.789,E2 9154.789} C_VEL
LIN {X 0,Y 425.403,Z 843.44,A -85,B 0,C 180,E1 9161.383,E2 9161.383} C_VEL
LIN {X 0,Y 425.665,Z 843.44,A -85,B 0,C 180,E1 9167.72,E2 9167.72} C_VEL
LIN {X 0,Y 425.82,Z 843.44,A -85,B 0,C 180,E1 9173.898,E2 9173.898} C_VEL
LIN {X 0,Y 426.065,Z 843.44,A -85,B 0,C 180,E1 9180,E2 9180} C_VEL
LIN {X 0,Y 425.749,Z 843.44,A -85,B 0,C 180,E1 9187.058,E2 9187.058} C_VEL
LIN {X 0,Y 425.565,Z 843.44,A -85,B 0,C 180,E1 9192.283,E2 9192.283} C_VEL
LIN {X 0,Y 425.323,Z 843.44,A -85,B 0,C 180,E1 9198.621,E2 9198.621} C_VEL
LIN {X 0,Y 425.125,Z 843.44,A -85,B 0,C 180,E1 9205.21,E2 9205.21} C_VEL
LIN {X 0,Y 424.894,Z 843.44,A -85,B 0,C 180,E1 9212.189,E2 9212.189} C_VEL
LIN {X 0,Y 424.911,Z 843.979,A -85,B 0,C 180,E1 9217.666,E2 9217.666} C_VEL
LIN {X 0,Y 427.646,Z 849.373,A -85,B 0,C 180,E1 9218.276,E2 9218.276} C_VEL
LIN {X 0,Y 448.246,Z 881.814,A -85,B 0,C 180,E1 9222.247,E2 9222.247} C_VEL
LIN {X 0,Y 464.425,Z 913.551,A -85,B 0,C 180,E1 9225.391,E2 9225.391} C_VEL
LIN {X 0,Y 460.208,Z 954.789,A -85,B 0,C 180,E1 9227.011,E2 9227.011} C_VEL
LIN {X 0,Y 454.673,Z 993.951,A -85,B 0,C 180,E1 9229.306,E2 9229.306} C_VEL
LIN {X 0,Y 448.014,Z 1032.639,A -85,B 0,C 180,E1 9232.476,E2 9232.476} C_VEL
LIN {X 0,Y 441.279,Z 1069.066,A -85,B 0,C 180,E1 9236.536,E2 9236.536} C_VEL
LIN {X 0,Y 435.319,Z 1100.955,A -85,B 0,C 180,E1 9241.278,E2 9241.278} C_VEL
LIN {X 0,Y 434.359,Z 1106.178,A -85,B 0,C 180,E1 9242.206,E2 9242.206} C_VEL
LIN {X 0,Y 428.812,Z 1116.461,A -85,B 0,C 180,E1 9243.947,E2 9243.947} C_VEL
LIN {X 0,Y 423.436,Z 1125.993,A -85,B 0,C 180,E1 9245.796,E2 9245.796} C_VEL
LIN {X 0,Y 420.391,Z 1147.319,A -85,B 0,C 180,E1 9251.519,E2 9251.519} C_VEL
LIN {X 0,Y 418.945,Z 1161.409,A -85,B 0,C 180,E1 9257.003,E2 9257.003} C_VEL
LIN {X 0,Y 418.28,Z 1170.558,A -85,B 0,C 180,E1 9262.597,E2 9262.597} C_VEL
LIN {X 0,Y 418.158,Z 1174.659,A -85,B 0,C 180,E1 9267.932,E2 9267.932} C_VEL
LIN {X 0,Y 418.365,Z 1174.659,A -85,B 0,C 180,E1 9272.067,E2 9272.067} C_VEL
LIN {X 0,Y 418.304,Z 1170.526,A -85,B 0,C 180,E1 9277.431,E2 9277.431} C_VEL
LIN {X 0,Y 418.919,Z 1161.433,A -85,B 0,C 180,E1 9282.987,E2 9282.987} C_VEL
LIN {X 0,Y 420.409,Z 1147.459,A -85,B 0,C 180,E1 9288.436,E2 9288.436} C_VEL
LIN {X 0,Y 423.298,Z 1126.755,A -85,B 0,C 180,E1 9294.028,E2 9294.028} C_VEL
LIN {X 0,Y 428.101,Z 1100.322,A -85,B 0,C 180,E1 9299.315,E2 9299.315} C_VEL
LIN {X 0,Y 434.363,Z 1068.855,A -85,B 0,C 180,E1 9304.053,E2 9304.053} C_VEL
LIN {X 0,Y 441.616,Z 1032.049,A -85,B 0,C 180,E1 9308.197,E2 9308.197} C_VEL
LIN {X 0,Y 448.529,Z 993.686,A -85,B 0,C 180,E1 9311.368,E2 9311.368} C_VEL
LIN {X 0,Y 454.518,Z 953.643,A -85,B 0,C 180,E1 9313.719,E2 9313.719} C_VEL
LIN {X 0,Y 458.177,Z 915.951,A -85,B 0,C 180,E1 9315.272,E2 9315.272} C_VEL
LIN {X 0,Y 440.688,Z 881.888,A -85,B 0,C 180,E1 9318.838,E2 9318.838} C_VEL
LIN {X 0,Y 423.27,Z 854.812,A -85,B 0,C 180,E1 9322.338,E2 9322.338} C_VEL
LIN {X 0,Y 419.247,Z 848.967,A -85,B 0,C 180,E1 9323.212,E2 9323.212} C_VEL
LIN {X 0,Y 416.919,Z 843.44,A -85,B 0,C 180,E1 9323.86,E2 9323.86} C_VEL
LIN {X 0,Y 417.035,Z 843.44,A -85,B 0,C 180,E1 9330.277,E2 9330.277} C_VEL
LIN {X 0,Y 417.23,Z 843.44,A -85,B 0,C 180,E1 9336.557,E2 9336.557} C_VEL
LIN {X 0,Y 417.438,Z 843.44,A -85,B 0,C 180,E1 9343.191,E2 9343.191} C_VEL
LIN {X 0,Y 417.598,Z 843.44,A -85,B 0,C 180,E1 9349.591,E2 9349.591} C_VEL
LIN {X 0,Y 417.958,Z 843.44,A -85,B 0,C 180,E1 9355.859,E2 9355.859} C_VEL
LIN {X 0,Y 418.043,Z 843.44,A -85,B 0,C 180,E1 9362.068,E2 9362.068} C_VEL
LIN {X 0,Y 417.786,Z 843.44,A -85,B 0,C 180,E1 9368.306,E2 9368.306} C_VEL
LIN {X 0,Y 417.594,Z 843.44,A -85,B 0,C 180,E1 9374.651,E2 9374.651} C_VEL
LIN {X 0,Y 417.34,Z 843.44,A -85,B 0,C 180,E1 9381.196,E2 9381.196} C_VEL
LIN {X 0,Y 417.083,Z 843.44,A -85,B 0,C 180,E1 9388.055,E2 9388.055} C_VEL
LIN {X 0,Y 417.048,Z 843.44,A -85,B 0,C 180,E1 9395.374,E2 9395.374} C_VEL
LIN {X 0,Y 417.071,Z 844.116,A -85,B 0,C 180,E1 9396.735,E2 9396.735} C_VEL
LIN {X 0,Y 419.767,Z 849.43,A -85,B 0,C 180,E1 9397.377,E2 9397.377} C_VEL
LIN {X 0,Y 438.434,Z 879.009,A -85,B 0,C 180,E1 9401.41,E2 9401.41} C_VEL
LIN {X 0,Y 454.948,Z 913.148,A -85,B 0,C 180,E1 9405.32,E2 9405.32} C_VEL
LIN {X 0,Y 456.256,Z 919.119,A -85,B 0,C 180,E1 9405.844,E2 9405.844} C_VEL
LIN {X 0,Y 450.807,Z 958.252,A -85,B 0,C 180,E1 9407.973,E2 9407.973} C_VEL
LIN {X 0,Y 443.939,Z 996.798,A -85,B 0,C 180,E1 9410.95,E2 9410.95} C_VEL
LIN {X 0,Y 437.01,Z 1031.765,A -85,B 0,C 180,E1 9414.663,E2 9414.663} C_VEL
LIN {X 0,Y 430.493,Z 1062.712,A -85,B 0,C 180,E1 9419.032,E2 9419.032} C_VEL
LIN {X 0,Y 424.971,Z 1090.209,A -85,B 0,C 180,E1 9424.216,E2 9424.216} C_VEL
LIN {X 0,Y 421.312,Z 1111.316,A -85,B 0,C 180,E1 9429.56,E2 9429.56} C_VEL
LIN {X 0,Y 419.254,Z 1128.002,A -85,B 0,C 180,E1 9435.407,E2 9435.407} C_VEL
LIN {X 0,Y 418.412,Z 1138.032,A -85,B 0,C 180,E1 9440.66,E2 9440.66} C_VEL
LIN {X 0,Y 418.2,Z 1143.664,A -85,B 0,C 180,E1 9445.861,E2 9445.861} C_VEL
LIN {X 0,Y 418.212,Z 1144.998,A -85,B 0,C 180,E1 9450,E2 9450} C_VEL
LIN {X 0,Y 418.231,Z 1143.605,A -85,B 0,C 180,E1 9454.138,E2 9454.138} C_VEL
LIN {X 0,Y 418.476,Z 1137.899,A -85,B 0,C 180,E1 9459.338,E2 9459.338} C_VEL
LIN {X 0,Y 419.254,Z 1127.776,A -85,B 0,C 180,E1 9464.593,E2 9464.593} C_VEL
LIN {X 0,Y 421.24,Z 1111.017,A -85,B 0,C 180,E1 9470.443,E2 9470.443} C_VEL
LIN {X 0,Y 425.243,Z 1088.596,A -85,B 0,C 180,E1 9476.049,E2 9476.049} C_VEL
LIN {X 0,Y 430.855,Z 1060.876,A -85,B 0,C 180,E1 9481.172,E2 9481.172} C_VEL
LIN {X 0,Y 437.611,Z 1028.978,A -85,B 0,C 180,E1 9485.584,E2 9485.584} C_VEL
LIN {X 0,Y 444.546,Z 994.3,A -85,B 0,C 180,E1 9489.179,E2 9489.179} C_VEL
LIN {X 0,Y 451.232,Z 956.04,A -85,B 0,C 180,E1 9492.077,E2 9492.077} C_VEL
LIN {X 0,Y 455.949,Z 916.377,A -85,B 0,C 180,E1 9494.267,E2 9494.267} C_VEL
LIN {X 0,Y 440.628,Z 882.868,A -85,B 0,C 180,E1 9498.021,E2 9498.021} C_VEL
LIN {X 0,Y 423.428,Z 855.078,A -85,B 0,C 180,E1 9501.719,E2 9501.719} C_VEL
LIN {X 0,Y 417.068,Z 844.706,A -85,B 0,C 180,E1 9503.145,E2 9503.145} C_VEL
LIN {X 0,Y 416.93,Z 843.44,A -85,B 0,C 180,E1 9503.278,E2 9503.278} C_VEL
LIN {X 0,Y 417.032,Z 843.44,A -85,B 0,C 180,E1 9510.276,E2 9510.276} C_VEL
LIN {X 0,Y 417.224,Z 843.44,A -85,B 0,C 180,E1 9516.558,E2 9516.558} C_VEL
LIN {X 0,Y 417.569,Z 843.44,A -85,B 0,C 180,E1 9523.197,E2 9523.197} C_VEL
LIN {X 0,Y 417.762,Z 843.44,A -85,B 0,C 180,E1 9529.596,E2 9529.596} C_VEL
LIN {X 0,Y 418.008,Z 843.44,A -85,B 0,C 180,E1 9535.86,E2 9535.86} C_VEL
LIN {X 0,Y 418.195,Z 843.44,A -85,B 0,C 180,E1 9542.068,E2 9542.068} C_VEL
LIN {X 0,Y 417.8,Z 843.44,A -85,B 0,C 180,E1 9548.307,E2 9548.307} C_VEL
LIN {X 0,Y 417.537,Z 843.44,A -85,B 0,C 180,E1 9554.654,E2 9554.654} C_VEL
LIN {X 0,Y 417.338,Z 843.44,A -85,B 0,C 180,E1 9561.197,E2 9561.197} C_VEL
LIN {X 0,Y 417.053,Z 843.44,A -85,B 0,C 180,E1 9568.058,E2 9568.058} C_VEL
LIN {X 0,Y 416.929,Z 843.44,A -85,B 0,C 180,E1 9575.386,E2 9575.386} C_VEL
LIN {X 0,Y 416.92,Z 843.44,A -85,B 0,C 180,E1 9576.213,E2 9576.213} C_VEL
LIN {X 0,Y 419.201,Z 848.951,A -85,B 0,C 180,E1 9576.792,E2 9576.792} C_VEL
LIN {X 0,Y 422.663,Z 854.01,A -85,B 0,C 180,E1 9577.546,E2 9577.546} C_VEL
LIN {X 0,Y 439.831,Z 880.404,A -85,B 0,C 180,E1 9581,E2 9581} C_VEL
LIN {X 0,Y 457.63,Z 914.669,A -85,B 0,C 180,E1 9584.608,E2 9584.608} C_VEL
LIN {X 0,Y 458.439,Z 919.264,A -85,B 0,C 180,E1 9584.902,E2 9584.902} C_VEL
LIN {X 0,Y 453.624,Z 959.688,A -85,B 0,C 180,E1 9586.582,E2 9586.582} C_VEL
LIN {X 0,Y 447.749,Z 998.143,A -85,B 0,C 180,E1 9588.96,E2 9588.96} C_VEL
LIN {X 0,Y 440.935,Z 1035.352,A -85,B 0,C 180,E1 9592.13,E2 9592.13} C_VEL
LIN {X 0,Y 434.379,Z 1068.854,A -85,B 0,C 180,E1 9595.947,E2 9595.947} C_VEL
LIN {X 0,Y 428.158,Z 1100.332,A -85,B 0,C 180,E1 9600.691,E2 9600.691} C_VEL
LIN {X 0,Y 423.436,Z 1125.993,A -85,B 0,C 180,E1 9605.796,E2 9605.796} C_VEL
LIN {X 0,Y 418.33,Z 1134.709,A -85,B 0,C 180,E1 9607.748,E2 9607.748} C_VEL
LIN {X 0,Y 413.294,Z 1142.59,A -85,B 0,C 180,E1 9609.803,E2 9609.803} C_VEL
LIN {X 0,Y 411.289,Z 1159.085,A -85,B 0,C 180,E1 9615.674,E2 9615.674} C_VEL
LIN {X 0,Y 410.441,Z 1169.517,A -85,B 0,C 180,E1 9621.543,E2 9621.543} C_VEL
LIN {X 0,Y 410.284,Z 1173.636,A -85,B 0,C 180,E1 9625.782,E2 9625.782} C_VEL
LIN {X 0,Y 410.312,Z 1175,A -85,B 0,C 180,E1 9630,E2 9630} C_VEL
LIN {X 0,Y 410.346,Z 1173.636,A -85,B 0,C 180,E1 9634.218,E2 9634.218} C_VEL
LIN {X 0,Y 410.533,Z 1167.965,A -85,B 0,C 180,E1 9639.521,E2 9639.521} C_VEL
LIN {X 0,Y 411.33,Z 1157.817,A -85,B 0,C 180,E1 9644.881,E2 9644.881} C_VEL
LIN {X 0,Y 413.62,Z 1140.464,A -85,B 0,C 180,E1 9650.837,E2 9650.837} C_VEL
LIN {X 0,Y 417.633,Z 1117.132,A -85,B 0,C 180,E1 9656.561,E2 9656.561} C_VEL
LIN {X 0,Y 423.39,Z 1088.077,A -85,B 0,C 180,E1 9661.849,E2 9661.849} C_VEL
LIN {X 0,Y 430.372,Z 1054.888,A -85,B 0,C 180,E1 9666.381,E2 9666.381} C_VEL
LIN {X 0,Y 437.828,Z 1018.364,A -85,B 0,C 180,E1 9670.097,E2 9670.097} C_VEL
LIN {X 0,Y 444.922,Z 978.688,A -85,B 0,C 180,E1 9673.037,E2 9673.037} C_VEL
LIN {X 0,Y 450.98,Z 935.771,A -85,B 0,C 180,E1 9675.212,E2 9675.212} C_VEL
LIN {X 0,Y 452.341,Z 919.32,A -85,B 0,C 180,E1 9675.864,E2 9675.864} C_VEL
LIN {X 0,Y 435.294,Z 885.348,A -85,B 0,C 180,E1 9679.546,E2 9679.546} C_VEL
LIN {X 0,Y 416.15,Z 855.711,A -85,B 0,C 180,E1 9683.59,E2 9683.59} C_VEL
LIN {X 0,Y 411.002,Z 848.64,A -85,B 0,C 180,E1 9684.774,E2 9684.774} C_VEL
LIN {X 0,Y 408.954,Z 843.44,A -85,B 0,C 180,E1 9685.462,E2 9685.462} C_VEL
LIN {X 0,Y 409.135,Z 843.44,A -85,B 0,C 180,E1 9692.276,E2 9692.276} C_VEL
LIN {X 0,Y 409.382,Z 843.44,A -85,B 0,C 180,E1 9698.371,E2 9698.371} C_VEL
LIN {X 0,Y 409.505,Z 843.44,A -85,B 0,C 180,E1 9705.052,E2 9705.052} C_VEL
LIN {X 0,Y 409.822,Z 843.44,A -85,B 0,C 180,E1 9711.531,E2 9711.531} C_VEL
LIN {X 0,Y 410.284,Z 843.44,A -85,B 0,C 180,E1 9717.892,E2 9717.892} C_VEL
LIN {X 0,Y 410.086,Z 843.44,A -85,B 0,C 180,E1 9724.22,E2 9724.22} C_VEL
LIN {X 0,Y 409.816,Z 843.44,A -85,B 0,C 180,E1 9730.609,E2 9730.609} C_VEL
LIN {X 0,Y 409.561,Z 843.44,A -85,B 0,C 180,E1 9737.142,E2 9737.142} C_VEL
LIN {X 0,Y 409.283,Z 843.44,A -85,B 0,C 180,E1 9743.925,E2 9743.925} C_VEL
LIN {X 0,Y 409.115,Z 843.44,A -85,B 0,C 180,E1 9751.089,E2 9751.089} C_VEL
LIN {X 0,Y 409.154,Z 843.824,A -85,B 0,C 180,E1 9755.2,E2 9755.2} C_VEL
LIN {X 0,Y 411.64,Z 849.21,A -85,B 0,C 180,E1 9755.85,E2 9755.85} C_VEL
LIN {X 0,Y 428.408,Z 874.787,A -85,B 0,C 180,E1 9759.673,E2 9759.673} C_VEL
LIN {X 0,Y 444.164,Z 905.481,A -85,B 0,C 180,E1 9763.477,E2 9763.477} C_VEL
LIN {X 0,Y 450.452,Z 920.653,A -85,B 0,C 180,E1 9765.199,E2 9765.199} C_VEL
LIN {X 0,Y 444.893,Z 958.544,A -85,B 0,C 180,E1 9767.283,E2 9767.283} C_VEL
LIN {X 0,Y 437.872,Z 996.467,A -85,B 0,C 180,E1 9770.23,E2 9770.23} C_VEL
LIN {X 0,Y 430.686,Z 1030.766,A -85,B 0,C 180,E1 9773.869,E2 9773.869} C_VEL
LIN {X 0,Y 423.545,Z 1062.954,A -85,B 0,C 180,E1 9778.455,E2 9778.455} C_VEL
LIN {X 0,Y 417.581,Z 1090.513,A -85,B 0,C 180,E1 9783.725,E2 9783.725} C_VEL
LIN {X 0,Y 413.706,Z 1111.618,A -85,B 0,C 180,E1 9789.167,E2 9789.167} C_VEL
LIN {X 0,Y 411.47,Z 1128.103,A -85,B 0,C 180,E1 9795.124,E2 9795.124} C_VEL
LIN {X 0,Y 410.523,Z 1138.031,A -85,B 0,C 180,E1 9800.479,E2 9800.479} C_VEL
LIN {X 0,Y 410.29,Z 1143.663,A -85,B 0,C 180,E1 9805.781,E2 9805.781} C_VEL
LIN {X 0,Y 410.311,Z 1144.998,A -85,B 0,C 180,E1 9810,E2 9810} C_VEL
LIN {X 0,Y 410.324,Z 1143.606,A -85,B 0,C 180,E1 9814.218,E2 9814.218} C_VEL
LIN {X 0,Y 410.577,Z 1137.9,A -85,B 0,C 180,E1 9819.52,E2 9819.52} C_VEL
LIN {X 0,Y 411.56,Z 1126.591,A -85,B 0,C 180,E1 9825.416,E2 9825.416} C_VEL
LIN {X 0,Y 413.666,Z 1111.323,A -85,B 0,C 180,E1 9830.834,E2 9830.834} C_VEL
LIN {X 0,Y 417.927,Z 1088.906,A -85,B 0,C 180,E1 9836.54,E2 9836.54} C_VEL
LIN {X 0,Y 423.884,Z 1061.282,A -85,B 0,C 180,E1 9841.728,E2 9841.728} C_VEL
LIN {X 0,Y 430.998,Z 1029.462,A -85,B 0,C 180,E1 9846.192,E2 9846.192} C_VEL
LIN {X 0,Y 438.39,Z 994.283,A -85,B 0,C 180,E1 9849.874,E2 9849.874} C_VEL
LIN {X 0,Y 445.553,Z 955.173,A -85,B 0,C 180,E1 9852.841,E2 9852.841} C_VEL
LIN {X 0,Y 450.354,Z 920.666,A -85,B 0,C 180,E1 9854.721,E2 9854.721} C_VEL
LIN {X 0,Y 435.539,Z 887.384,A -85,B 0,C 180,E1 9858.585,E2 9858.585} C_VEL
LIN {X 0,Y 418.836,Z 859.924,A -85,B 0,C 180,E1 9862.379,E2 9862.379} C_VEL
LIN {X 0,Y 411.736,Z 849.427,A -85,B 0,C 180,E1 9864.019,E2 9864.019} C_VEL
LIN {X 0,Y 409.117,Z 844.692,A -85,B 0,C 180,E1 9864.674,E2 9864.674} C_VEL
LIN {X 0,Y 409.003,Z 843.44,A -85,B 0,C 180,E1 9864.825,E2 9864.825} C_VEL
LIN {X 0,Y 409.114,Z 843.44,A -85,B 0,C 180,E1 9872.281,E2 9872.281} C_VEL
LIN {X 0,Y 409.375,Z 843.44,A -85,B 0,C 180,E1 9878.371,E2 9878.371} C_VEL
LIN {X 0,Y 409.737,Z 843.44,A -85,B 0,C 180,E1 9885.061,E2 9885.061} C_VEL
LIN {X 0,Y 409.901,Z 843.44,A -85,B 0,C 180,E1 9891.533,E2 9891.533} C_VEL
LIN {X 0,Y 410.135,Z 843.44,A -85,B 0,C 180,E1 9897.892,E2 9897.892} C_VEL
LIN {X 0,Y 410.044,Z 843.44,A -85,B 0,C 180,E1 9904.221,E2 9904.221} C_VEL
LIN {X 0,Y 409.769,Z 843.44,A -85,B 0,C 180,E1 9910.61,E2 9910.61} C_VEL
LIN {X 0,Y 409.529,Z 843.44,A -85,B 0,C 180,E1 9917.144,E2 9917.144} C_VEL
LIN {X 0,Y 409.3,Z 843.44,A -85,B 0,C 180,E1 9923.925,E2 9923.925} C_VEL
LIN {X 0,Y 409.005,Z 843.44,A -85,B 0,C 180,E1 9931.098,E2 9931.098} C_VEL
LIN {X 0,Y 408.988,Z 843.638,A -85,B 0,C 180,E1 9934.696,E2 9934.696} C_VEL
LIN {X 0,Y 411.199,Z 848.851,A -85,B 0,C 180,E1 9935.287,E2 9935.287} C_VEL
LIN {X 0,Y 414.378,Z 853.4,A -85,B 0,C 180,E1 9936.028,E2 9936.028} C_VEL
LIN {X 0,Y 430.795,Z 877.987,A -85,B 0,C 180,E1 9939.541,E2 9939.541} C_VEL
LIN {X 0,Y 447.836,Z 909.257,A -85,B 0,C 180,E1 9943.107,E2 9943.107} C_VEL
LIN {X 0,Y 452.645,Z 921.167,A -85,B 0,C 180,E1 9944.257,E2 9944.257} C_VEL
LIN {X 0,Y 447.505,Z 961.651,A -85,B 0,C 180,E1 9945.993,E2 9945.993} C_VEL
LIN {X 0,Y 441.483,Z 998.807,A -85,B 0,C 180,E1 9948.341,E2 9948.341} C_VEL
LIN {X 0,Y 434.427,Z 1035.26,A -85,B 0,C 180,E1 9951.487,E2 9951.487} C_VEL
LIN {X 0,Y 427.492,Z 1068.761,A -85,B 0,C 180,E1 9955.356,E2 9955.356} C_VEL
LIN {X 0,Y 420.942,Z 1100.195,A -85,B 0,C 180,E1 9960.172,E2 9960.172} C_VEL
LIN {X 0,Y 415.719,Z 1126.851,A -85,B 0,C 180,E1 9965.61,E2 9965.61} C_VEL
LIN {X 0,Y 413.294,Z 1142.59,A -85,B 0,C 180,E1 9969.803,E2 9969.803} C_VEL
LIN {X 0,Y 408.384,Z 1149.65,A -85,B 0,C 180,E1 9971.94,E2 9971.94} C_VEL
LIN {X 0,Y 403.787,Z 1155.866,A -85,B 0,C 180,E1 9974.164,E2 9974.164} C_VEL
LIN {X 0,Y 402.766,Z 1166.249,A -85,B 0,C 180,E1 9979.203,E2 9979.203} C_VEL
LIN {X 0,Y 402.422,Z 1171.925,A -85,B 0,C 180,E1 9983.541,E2 9983.541} C_VEL
LIN {X 0,Y 402.377,Z 1174.659,A -85,B 0,C 180,E1 9987.851,E2 9987.851} C_VEL
LIN {X 0,Y 402.565,Z 1174.659,A -85,B 0,C 180,E1 9992.148,E2 9992.148} C_VEL
LIN {X 0,Y 402.468,Z 1171.314,A -85,B 0,C 180,E1 9997.012,E2 9997.012} C_VEL
LIN {X 0,Y 403.127,Z 1162.275,A -85,B 0,C 180,E1 10002.979,E2 10002.979} C_VEL
LIN {X 0,Y 404.822,Z 1147.522,A -85,B 0,C 180,E1 10008.935,E2 10008.935} C_VEL
LIN {X 0,Y 408.038,Z 1127.337,A -85,B 0,C 180,E1 10014.67,E2 10014.67} C_VEL
LIN {X 0,Y 413.415,Z 1101.36,A -85,B 0,C 180,E1 10020.125,E2 10020.125} C_VEL
LIN {X 0,Y 420.079,Z 1071.202,A -85,B 0,C 180,E1 10024.9,E2 10024.9} C_VEL
LIN {X 0,Y 427.502,Z 1037.67,A -85,B 0,C 180,E1 10028.91,E2 10028.91} C_VEL
LIN {X 0,Y 434.746,Z 1002.188,A -85,B 0,C 180,E1 10032.094,E2 10032.094} C_VEL
LIN {X 0,Y 441.527,Z 963.021,A -85,B 0,C 180,E1 10034.646,E2 10034.646} C_VEL
LIN {X 0,Y 446.343,Z 922.217,A -85,B 0,C 180,E1 10036.518,E2 10036.518} C_VEL
LIN {X 0,Y 430.451,Z 889.938,A -85,B 0,C 180,E1 10040.161,E2 10040.161} C_VEL
LIN {X 0,Y 412.552,Z 861.818,A -85,B 0,C 180,E1 10044.09,E2 10044.09} C_VEL
LIN {X 0,Y 403.596,Z 849.216,A -85,B 0,C 180,E1 10046.259,E2 10046.259} C_VEL
LIN {X 0,Y 401.129,Z 844.453,A -85,B 0,C 180,E1 10046.937,E2 10046.937} C_VEL
LIN {X 0,Y 401.048,Z 843.44,A -85,B 0,C 180,E1 10047.143,E2 10047.143} C_VEL
LIN {X 0,Y 401.228,Z 843.44,A -85,B 0,C 180,E1 10054.507,E2 10054.507} C_VEL
LIN {X 0,Y 401.514,Z 843.44,A -85,B 0,C 180,E1 10060.23,E2 10060.23} C_VEL
LIN {X 0,Y 401.707,Z 843.44,A -85,B 0,C 180,E1 10067.606,E2 10067.606} C_VEL
LIN {X 0,Y 402.123,Z 843.44,A -85,B 0,C 180,E1 10073.536,E2 10073.536} C_VEL
LIN {X 0,Y 402.332,Z 843.44,A -85,B 0,C 180,E1 10080,E2 10080} C_VEL
LIN {X 0,Y 402.093,Z 843.44,A -85,B 0,C 180,E1 10086.464,E2 10086.464} C_VEL
LIN {X 0,Y 401.838,Z 843.44,A -85,B 0,C 180,E1 10093.021,E2 10093.021} C_VEL
LIN {X 0,Y 401.481,Z 843.44,A -85,B 0,C 180,E1 10100.006,E2 10100.006} C_VEL
LIN {X 0,Y 401.25,Z 843.44,A -85,B 0,C 180,E1 10106.825,E2 10106.825} C_VEL
LIN {X 0,Y 401.28,Z 844.094,A -85,B 0,C 180,E1 10113.567,E2 10113.567} C_VEL
LIN {X 0,Y 403.863,Z 849.368,A -85,B 0,C 180,E1 10114.284,E2 10114.284} C_VEL
LIN {X 0,Y 406.906,Z 853.729,A -85,B 0,C 180,E1 10115.046,E2 10115.046} C_VEL
LIN {X 0,Y 422.374,Z 877.57,A -85,B 0,C 180,E1 10118.778,E2 10118.778} C_VEL
LIN {X 0,Y 437.753,Z 907.336,A -85,B 0,C 180,E1 10122.671,E2 10122.671} C_VEL
LIN {X 0,Y 444.431,Z 924.093,A -85,B 0,C 180,E1 10124.62,E2 10124.62} C_VEL
LIN {X 0,Y 438.308,Z 963.016,A -85,B 0,C 180,E1 10126.86,E2 10126.86} C_VEL
LIN {X 0,Y 431.091,Z 999.517,A -85,B 0,C 180,E1 10129.806,E2 10129.806} C_VEL
LIN {X 0,Y 423.736,Z 1032.779,A -85,B 0,C 180,E1 10133.444,E2 10133.444} C_VEL
LIN {X 0,Y 416.336,Z 1064.33,A -85,B 0,C 180,E1 10138.054,E2 10138.054} C_VEL
LIN {X 0,Y 410.308,Z 1090.814,A -85,B 0,C 180,E1 10143.222,E2 10143.222} C_VEL
LIN {X 0,Y 406.132,Z 1111.919,A -85,B 0,C 180,E1 10148.76,E2 10148.76} C_VEL
LIN {X 0,Y 403.7,Z 1128.403,A -85,B 0,C 180,E1 10154.831,E2 10154.831} C_VEL
LIN {X 0,Y 402.647,Z 1138.165,A -85,B 0,C 180,E1 10160.291,E2 10160.291} C_VEL
LIN {X 0,Y 402.388,Z 1143.662,A -85,B 0,C 180,E1 10165.698,E2 10165.698} C_VEL
LIN {X 0,Y 402.421,Z 1144.998,A -85,B 0,C 180,E1 10170,E2 10170} C_VEL
LIN {X 0,Y 402.424,Z 1143.607,A -85,B 0,C 180,E1 10174.301,E2 10174.301} C_VEL
LIN {X 0,Y 402.689,Z 1138.039,A -85,B 0,C 180,E1 10179.708,E2 10179.708} C_VEL
LIN {X 0,Y 403.678,Z 1128.193,A -85,B 0,C 180,E1 10185.169,E2 10185.169} C_VEL
LIN {X 0,Y 406.118,Z 1111.63,A -85,B 0,C 180,E1 10191.24,E2 10191.24} C_VEL
LIN {X 0,Y 410.637,Z 1089.217,A -85,B 0,C 180,E1 10197.049,E2 10197.049} C_VEL
LIN {X 0,Y 416.9,Z 1061.943,A -85,B 0,C 180,E1 10202.261,E2 10202.261} C_VEL
LIN {X 0,Y 424.444,Z 1029.773,A -85,B 0,C 180,E1 10206.842,E2 10206.842} C_VEL
LIN {X 0,Y 432.244,Z 994.6,A -85,B 0,C 180,E1 10210.557,E2 10210.557} C_VEL
LIN {X 0,Y 439.571,Z 956.341,A -85,B 0,C 180,E1 10213.493,E2 10213.493} C_VEL
LIN {X 0,Y 444.221,Z 923.348,A -85,B 0,C 180,E1 10215.362,E2 10215.362} C_VEL
LIN {X 0,Y 429.538,Z 890.094,A -85,B 0,C 180,E1 10219.384,E2 10219.384} C_VEL
